	    REGION 180

	        REGION Displacement
	            #sFB_Displacement180(#sUDT_Interface_180);
	        END_REGION

	        REGION Conveyor

	            #sUDT_Handshake_180.RTR := TRUE;

	            #sFB_Conveyor_080(iUDT_ConveyorConfiguration := #iqUDT_Configuration."180".Conveyor,
	                              idi_PECEoSDistance := 0,
	                              idi_PECBoSDistance := 0,
	                              ii_ExternalSpeed := 0,
	                              ix_SafetyOk := #ix_SafetyOk,
	                              ix_24vOk := #ix_24vOk,
	                              ix_400vOk := #ix_400vOk,
	                              ix_HardwareOk := TRUE,
	                              ix_PECEoS := TRUE,
	                              ix_PECBoS := TRUE,
	                              ix_ReverseDirection := FALSE,
	                              ix_ExternalRequestDieBack := FALSE,
	                              ix_ExternalRequestHold := #sx_Hold180,
	                              ix_ResetEnergySave := FALSE,
	                              qUDT_HMIStatus => #iqUDT_WorkstationStatus."180".Conveyor,
	                              qUDT_Status => #iqUDT_WorkstationCommonStatus."180",
	                              iqUDT_EquipmentControl := #iqUDT_EquipmentControl,
	                              iqUDT_ConveyorCommand := #iqUDT_WorkstationCommands."180".Conveyor,
	                              iqUDT_ConveyorInterface := #sUDT_Interface_180,
	                              iqUDT_HandShakeUp := #sUDT_HandshakeUp_180,
	                              iqUDT_HandShake := #sUDT_Handshake_180,
	                              iqUDT_Statistics := #iqUDT_WorkstationStatistics."180".Conveyor);

	        END_REGION

	        REGION MCO

	            #sFB_MCOConveyLinxAixController_180(iUDT_AixConfig := #iqUDT_Configuration."180".MCO_M01,
	                                                iUDT_AixInputsModule := #iUDT_MotorInput170,
	                                                ix_24vOk := #ix_24vOk,
	                                                ix_SimulationModeActive := "DB_Memory".Simulation,
	                                                ii_MotorPositionId := 2,
	                                                qUDT_HMIStatus => #iqUDT_WorkstationStatus."180".MCO_M01,
	                                                iqUDT_AixOutputsModule := #iqUDT_MotorOutput170,
	                                                iqUDT_ConveyorInterface := #sUDT_Interface_180,
	                                                iqUDT_MCOStatistics := #iqUDT_WorkstationStatistics."180".MCO_M01);
	        END_REGION

	    END_REGION
	END_IF;
	REGION 210

	    REGION Displacement
	        #sFB_Displacement210(#sUDT_Interface_210);
	    END_REGION

	    REGION Tracking

	        #sFB_Tracking_210(iUDT_ConveyorCommonConfiguration := #iqUDT_Configuration."210".Conveyor.Common,
	                          iqa_TrackingData := #sa_TrackingArray_210,
	                          iqUDT_ConveyorInterface := #sUDT_Interface_210,
	                          iqUDT_HandshakeUp := #sUDT_HandshakeUp_210,
	                          iqUDT_Handshake := #sUDT_Handshake_210);

	    END_REGION

	    REGION EoS

	        #sFB_PECUpdate_210(iUDT_PECUpdateConfiguration := #iqUDT_Configuration."210".PEC_EoS,
	                           iUDT_ConveyorCommonConfiguration := #iqUDT_Configuration."210".Conveyor.Common,
	                           ix_PEC := NOT #iUDT_MotorInput210.AllSensorPortInputs.LeftSensor,
	                           ix_TeachingMode := FALSE,
	                           qUDT_Status => #iqUDT_WorkstationStatus."210".PEC_EoS,
	                           iqUDT_ConveyorInterface := #sUDT_Interface_210,
	                           iqUDT_UnknownGINRange := #iqUDT_UnknownGINRange,
	                           iqUDT_FifoHeader := "DB_FIFOLostGIN".Header,
	                           iqUDT_Statistics := #iqUDT_WorkstationStatistics."210".PEC_EoS,
	                           iqa_TrackingData := #sa_TrackingArray_210,
	                           iqa_FifoData := "DB_FIFOLostGIN".Data);

	    END_REGION

	    REGION Conveyor

	        #sFB_Conveyor_210(iUDT_ConveyorConfiguration := #iqUDT_Configuration."210".Conveyor,
	                          idi_PECEoSDistance := #iqUDT_Configuration."210".PEC_EoS.Distance,
	                          idi_PECBoSDistance := 0,
	                          ii_ExternalSpeed := 0,
	                          ix_SafetyOk := #ix_SafetyOk,
	                          ix_24vOk := #ix_24vOk,
	                          ix_400vOk := #ix_400vOk,
	                          ix_HardwareOk := TRUE,
	                          ix_PECEoS := #iqUDT_WorkstationStatus."210".PEC_EoS.PEC,
	                          ix_PECBoS := TRUE,
	                          ix_ReverseDirection := FALSE,
	                          ix_ExternalRequestDieBack := FALSE,
	                          ix_ExternalRequestHold := #sx_ReleaseBinHoldLeft OR #sx_ReleaseBinHoldRight OR NOT #sUDT_Handshake_210.RTR,
	                          ix_ResetEnergySave := FALSE,
	                          qUDT_HMIStatus => #iqUDT_WorkstationStatus."210".Conveyor,
	                          qUDT_Status => #iqUDT_WorkstationCommonStatus."210",
	                          iqUDT_EquipmentControl := #iqUDT_EquipmentControl,
	                          iqUDT_ConveyorCommand := #iqUDT_WorkstationCommands."210".Conveyor,
	                          iqUDT_ConveyorInterface := #sUDT_Interface_210,
	                          iqUDT_HandShakeUp := #sUDT_HandshakeUp_210,
	                          iqUDT_HandShake := #sUDT_Handshake_210,
	                          iqUDT_Statistics := #iqUDT_WorkstationStatistics."210".Conveyor);

	    END_REGION

	    REGION MCO

	        #sFB_MCOConveyLinxAixController_210(iUDT_AixConfig := #iqUDT_Configuration."210".MCO_M01,
	                                            iUDT_AixInputsModule := #iUDT_MotorInput210,
	                                            ix_24vOk := #ix_24vOk,
	                                            ix_SimulationModeActive := "DB_Memory".Simulation,
	                                            ii_MotorPositionId := 1,
	                                            qUDT_HMIStatus => #iqUDT_WorkstationStatus."210".MCO_M01,
	                                            iqUDT_AixOutputsModule := #iqUDT_MotorOutput210,
	                                            iqUDT_ConveyorInterface := #sUDT_Interface_210,
	                                            iqUDT_MCOStatistics := #iqUDT_WorkstationStatistics."210".MCO_M01);
	    END_REGION

	END_REGION

	REGION 220

	    REGION Displacement
	        #sFB_Displacement220(#sUDT_Interface_220);
	    END_REGION

	    REGION Tracking

	        #sFB_Tracking_220(iUDT_ConveyorCommonConfiguration := #iqUDT_Configuration."220".Conveyor.Common,
	                          iqa_TrackingData := #sa_TrackingArray_220,
	                          iqUDT_ConveyorInterface := #sUDT_Interface_220,
	                          iqUDT_HandshakeUp := #sUDT_Handshake_210,
	                          iqUDT_Handshake := #sUDT_Handshake_220);

	    END_REGION

	    REGION EoS

	        #sFB_PECUpdate_220(iUDT_PECUpdateConfiguration := #iqUDT_Configuration."220".PEC_EoS,
	                           iUDT_ConveyorCommonConfiguration := #iqUDT_Configuration."220".Conveyor.Common,
	                           ix_PEC := NOT #iUDT_MotorInput210.AllSensorPortInputs.RightSensor,
	                           ix_TeachingMode := FALSE,
	                           qUDT_Status => #iqUDT_WorkstationStatus."220".PEC_EoS,
	                           iqUDT_ConveyorInterface := #sUDT_Interface_220,
	                           iqUDT_UnknownGINRange := #iqUDT_UnknownGINRange,
	                           iqUDT_FifoHeader := "DB_FIFOLostGIN".Header,
	                           iqUDT_Statistics := #iqUDT_WorkstationStatistics."220".PEC_EoS,
	                           iqa_TrackingData := #sa_TrackingArray_220,
	                           iqa_FifoData := "DB_FIFOLostGIN".Data);




	    END_REGION

	    REGION Conveyor

	        #sFB_Conveyor_220(iUDT_ConveyorConfiguration := #iqUDT_Configuration."220".Conveyor,
	                          idi_PECEoSDistance := #iqUDT_Configuration."220".PEC_EoS.Distance,
	                          idi_PECBoSDistance := 0,
	                          ii_ExternalSpeed := 0,
	                          ix_SafetyOk := #ix_SafetyOk,
	                          ix_24vOk := #ix_24vOk,
	                          ix_400vOk := #ix_400vOk,
	                          ix_HardwareOk := TRUE,
	                          ix_PECEoS := #iqUDT_WorkstationStatus."220".PEC_EoS.PEC,
	                          ix_PECBoS := TRUE,
	                          ix_ReverseDirection := FALSE,
	                          ix_ExternalRequestDieBack := FALSE,
	                          ix_ExternalRequestHold := #sx_Hold220 OR #sx_ReleaseBinHoldLeft OR #sx_ReleaseBinHoldRight,
	                          ix_ResetEnergySave := FALSE,
	                          qUDT_HMIStatus => #iqUDT_WorkstationStatus."220".Conveyor,
	                          qUDT_Status => #iqUDT_WorkstationCommonStatus."220",
	                          iqUDT_EquipmentControl := #iqUDT_EquipmentControl,
	                          iqUDT_ConveyorCommand := #iqUDT_WorkstationCommands."220".Conveyor,
	                          iqUDT_ConveyorInterface := #sUDT_Interface_220,
	                          iqUDT_HandShakeUp := #sUDT_Handshake_210,
	                          iqUDT_HandShake := #sUDT_Handshake_220,
	                          iqUDT_Statistics := #iqUDT_WorkstationStatistics."220".Conveyor);

	    END_REGION

	    REGION MCO

	        #sFB_MCOConveyLinxAixController_220(iUDT_AixConfig := #iqUDT_Configuration."220".MCO_M01,
	                                            iUDT_AixInputsModule := #iUDT_MotorInput210,
	                                            ix_24vOk := #ix_24vOk,
	                                            ix_SimulationModeActive := "DB_Memory".Simulation,
	                                            ii_MotorPositionId := 2,
	                                            qUDT_HMIStatus => #iqUDT_WorkstationStatus."220".MCO_M01,
	                                            iqUDT_AixOutputsModule := #iqUDT_MotorOutput210,
	                                            iqUDT_ConveyorInterface := #sUDT_Interface_220,
	                                            iqUDT_MCOStatistics := #iqUDT_WorkstationStatistics."220".MCO_M01);
	    END_REGION


	END_REGION

	REGION 230

	    REGION Displacement
	        #sFB_Displacement230(#sUDT_Interface_230);
	    END_REGION

	    REGION Tracking

	        #sFB_Tracking_230(iUDT_ConveyorCommonConfiguration := #iqUDT_Configuration."230".Conveyor.Common,
	                          iqa_TrackingData := #sa_TrackingArray_230,
	                          iqUDT_ConveyorInterface := #sUDT_Interface_230,
	                          iqUDT_HandshakeUp := #sUDT_Handshake_220,
	                          iqUDT_Handshake := #sUDT_Handshake_230);

	    END_REGION

	    REGION EoS

	        #sFB_PECUpdate_230(iUDT_PECUpdateConfiguration := #iqUDT_Configuration."230".PEC_EoS,
	                           iUDT_ConveyorCommonConfiguration := #iqUDT_Configuration."230".Conveyor.Common,
	                           ix_PEC := NOT #iUDT_MotorInput230.AllSensorPortInputs.LeftSensor,
	                           ix_TeachingMode := FALSE,
	                           qUDT_Status => #iqUDT_WorkstationStatus."230".PEC_EoS,
	                           iqUDT_ConveyorInterface := #sUDT_Interface_230,
	                           iqUDT_UnknownGINRange := #iqUDT_UnknownGINRange,
	                           iqUDT_FifoHeader := "DB_FIFOLostGIN".Header,
	                           iqUDT_Statistics := #iqUDT_WorkstationStatistics."230".PEC_EoS,
	                           iqa_TrackingData := #sa_TrackingArray_230,
	                           iqa_FifoData := "DB_FIFOLostGIN".Data);




	    END_REGION

	    REGION Conveyor
	        #sUDT_Handshake_230.RTR := #sUDT_Handshake_230.RTR OR #iqUDT_WorkstationStatus."230".PEC_EoS.PEC;
	        #sFB_Conveyor_230(iUDT_ConveyorConfiguration := #iqUDT_Configuration."230".Conveyor,
	                          idi_PECEoSDistance := #iqUDT_Configuration."230".PEC_EoS.Distance,
	                          idi_PECBoSDistance := 0,
	                          ii_ExternalSpeed := 0,
	                          ix_SafetyOk := #ix_SafetyOk,
	                          ix_24vOk := #ix_24vOk,
	                          ix_400vOk := #ix_400vOk,
	                          ix_HardwareOk := TRUE,
	                          ix_PECEoS := #iqUDT_WorkstationStatus."230".PEC_EoS.PEC,
	                          ix_PECBoS := TRUE,
	                          ix_ReverseDirection := FALSE,
	                          ix_ExternalRequestDieBack := FALSE,
	                          ix_ExternalRequestHold := #sx_Hold230 OR #sx_ReleaseBinHoldLeft OR #sx_ReleaseBinHoldRight,
	                          ix_ResetEnergySave := FALSE,
	                          qUDT_HMIStatus => #iqUDT_WorkstationStatus."230".Conveyor,
	                          qUDT_Status => #iqUDT_WorkstationCommonStatus."230",
	                          iqUDT_EquipmentControl := #iqUDT_EquipmentControl,
	                          iqUDT_ConveyorCommand := #iqUDT_WorkstationCommands."230".Conveyor,
	                          iqUDT_ConveyorInterface := #sUDT_Interface_230,
	                          iqUDT_HandShakeUp := #sUDT_Handshake_220,
	                          iqUDT_HandShake := #sUDT_Handshake_230,
	                          iqUDT_Statistics := #iqUDT_WorkstationStatistics."230".Conveyor);

	    END_REGION

	    REGION MCO

	        #sFB_MCOConveyLinxAixController_230(iUDT_AixConfig := #iqUDT_Configuration."230".MCO_M01,
	                                            iUDT_AixInputsModule := #iUDT_MotorInput230,
	                                            ix_24vOk := #ix_24vOk,
	                                            ix_SimulationModeActive := "DB_Memory".Simulation,
	                                            ii_MotorPositionId := 1,
	                                            qUDT_HMIStatus => #iqUDT_WorkstationStatus."230".MCO_M01,
	                                            iqUDT_AixOutputsModule := #iqUDT_MotorOutput230,
	                                            iqUDT_ConveyorInterface := #sUDT_Interface_230,
	                                            iqUDT_MCOStatistics := #iqUDT_WorkstationStatistics."230".MCO_M01);
	    END_REGION

	END_REGION

	REGION 240

	    REGION Displacement
	        #sFB_Displacement240(#sUDT_Interface_240);
	    END_REGION

	    REGION MCO

	        #sFB_MCOConveyLinxAixController_240(iUDT_AixConfig := #iqUDT_Configuration."240".MCO_M01,
	                                            iUDT_AixInputsModule := #iUDT_MotorInput240,
	                                            ii_PositionSetpoint := #iqUDT_RATPositioning240.Lower.EndPosition,
	                                            ix_24vOk := #ix_24vOk,
	                                            ix_SimulationModeActive := "DB_Memory".Simulation,
	                                            ii_MotorPositionId := 1,
	                                            ix_StartPositioning := #iqUDT_RATPositioning240.Lower.Start,
	                                            ix_ResetPosition := #iqUDT_RATPositioning240.Lower.ResetPosition,
	                                            qUDT_HMIStatus => #iqUDT_WorkstationStatus."240".MCO_M01,
	                                            qx_Positioned => #iqUDT_RATPositioning240.Lower.Done,
	                                            iqUDT_AixOutputsModule := #iqUDT_MotorOutput240,
	                                            iqUDT_ConveyorInterface := #sUDT_Interface_240,
	                                            iqUDT_MCOStatistics := #iqUDT_WorkstationStatistics."240".MCO_M01);
	    END_REGION

	END_REGION

	REGION 241

	    REGION Displacement
	        #sFB_Displacement241(#sUDT_Interface_241);
	    END_REGION

	    REGION RAT

	        #sFB_RightAngledTransfer_241(iUDT_Configuration := #iqUDT_Configuration."241".RightAngledTransfer,
	                                     iUDT_LowerConveyorConfiguration := #iqUDT_Configuration."240".Conveyor,
	                                     iUDT_UpperConveyorConfiguration := #iqUDT_Configuration."241".Conveyor,
	                                     iUDT_PECConfiguration := #iqUDT_Configuration."240".PEC_EoS,
	                                     ii_DestinationA := #si_240DestinationA,
	                                     ii_DestinationB := #si_240DestinationB,
	                                     ii_DestinationC := #si_240DestinationC,
	                                     ii_DestinationD := #si_240DestinationD,
	                                     ix_HardwareOk := TRUE,
	                                     ix_400vOk := #ix_400vOk,
	                                     ix_24vOk := #ix_24vOk,
	                                     ix_SafetyOk := #ix_SafetyOk,
	                                     ix_AirPressureOk := #ix_AirPressureOk,
	                                     ix_SectionIsDown := #ix_SectionisDown241,
	                                     ix_SectionIsUp := #ix_SectionisUp241,
	                                     ix_ConveyorAAuto := #iqUDT_WorkstationCommonStatus."230".AutoON,
	                                     ix_ConveyorBAuto := #iqUDT_WorkstationCommonStatus."250".AutoON,
	                                     ix_ConveyorCAuto := #iqUDT_WorkstationCommonStatus."141".AutoON,
	                                     ix_ConveyorDAuto := #iqUDT_WorkstationCommonStatus."041".AutoON,
	                                     ix_PEC := #iUDT_MotorInput240.AllSensorPortInputs.LeftSensor,
	                                     ix_ExternalReceiveRequestA := NOT #iqUDT_WorkstationStatus."230".PEC_EoS.PEC AND #sx_Enable2X0In,
	                                     ix_ExternalReceiveRequestB := false,
	                                     ix_ExternalReceiveRequestC := #sFB_RightAngledTransfer_141.qx_ExternalSendRequestC,
	                                     ix_ExternalReceiveRequestD := #sFB_RightAngledTransfer_041.qx_ExternalSendRequestD,
	                                     ix_PECInfeedA := #iqUDT_WorkstationStatus."230".PEC_EoS.PEC,
	                                     ix_PECInfeedC := #iqUDT_WorkstationStatus."140".PEC_EoS.PEC,
	                                     ix_PECInfeedD := #iqUDT_WorkstationStatus."040".PEC_EoS.PEC,
	                                     qUDT_HMIRATStatus => #iqUDT_WorkstationStatus."241".RightAngledTransfer,
	                                     qUDT_HMIConveyorStatus => #iqUDT_WorkstationStatus."240".Conveyor,
	                                     qUDT_HMIPECStatus => #iqUDT_WorkstationStatus."240".PEC_EoS,
	                                     qUDT_RATStatus => #iqUDT_WorkstationCommonStatus."241",
	                                     qUDT_ConveyorStatus => #iqUDT_WorkstationCommonStatus."240",
	                                     qx_PopupControl => #qx_PopupControl241,
	                                     iqUDT_EquipmentControl := #iqUDT_EquipmentControl,
	                                     iqUDT_RATCommand := #iqUDT_WorkstationCommands."241".RightAngledTransfer,
	                                     iqUDT_ConveyorCommand := #iqUDT_WorkstationCommands."240".Conveyor,
	                                     iqUDT_RATStatistics := #iqUDT_WorkstationStatistics."241".RightAngledTransfer,
	                                     iqUDT_ConveyorStatistics := #iqUDT_WorkstationStatistics."240".Conveyor,
	                                     iqUDT_PECStatistics := #iqUDT_WorkstationStatistics."240".PEC_EoS,
	                                     iqUDT_HandShakeConveyorA := #sUDT_Handshake_230,
	                                     iqUDT_HandShakeConveyorB := #sUDT_Handshake_240,
	                                     iqUDT_HandShakeConveyorC := #sUDT_Handshake_241,
	                                     iqUDT_HandShakeConveyorD := #sUDT_Handshake_041,
	                                     iqUDT_LowerConveyorInterface := #sUDT_Interface_240,
	                                     iqUDT_UpperConveyorInterface := #sUDT_Interface_241,
	                                     iqUDT_RATPositioning := #iqUDT_RATPositioning240,
	                                     iqUDT_BladeStopEoSInterface := #tUDT_DummyBladeStop,
	                                     iqUDT_BladeStopBoSInterface := #tUDT_DummyBladeStop);

	    END_REGION

	    REGION MCO

	        #sFB_MCOConveyLinxAixController_241(iUDT_AixConfig := #iqUDT_Configuration."241".MCO_M01,
	                                            iUDT_AixInputsModule := #iUDT_MotorInput240,
	                                            ii_PositionSetpoint := #iqUDT_RATPositioning240.Upper.EndPosition,
	                                            ix_24vOk := #ix_24vOk,
	                                            ix_SimulationModeActive := "DB_Memory".Simulation,
	                                            ii_MotorPositionId := 2,
	                                            ix_StartPositioning := #iqUDT_RATPositioning240.Upper.Start,
	                                            ix_ResetPosition := #iqUDT_RATPositioning240.Upper.ResetPosition,
	                                            qUDT_HMIStatus => #iqUDT_WorkstationStatus."241".MCO_M01,
	                                            qx_Positioned => #iqUDT_RATPositioning240.Upper.Done,
	                                            iqUDT_AixOutputsModule := #iqUDT_MotorOutput240,
	                                            iqUDT_ConveyorInterface := #sUDT_Interface_241,
	                                            iqUDT_MCOStatistics := #iqUDT_WorkstationStatistics."241".MCO_M01);
	    END_REGION

	END_REGION

	REGION 250

	    REGION Displacement
	        #sFB_Displacement250(#sUDT_Interface_250);
	    END_REGION

	    REGION Tracking

	        #sFB_Tracking_250(iUDT_ConveyorCommonConfiguration := #iqUDT_Configuration."250".Conveyor.Common,
	                          iqa_TrackingData := #sa_TrackingArray_250,
	                          iqUDT_ConveyorInterface := #sUDT_Interface_250,
	                          iqUDT_HandshakeUp := #sUDT_Handshake_240,
	                          iqUDT_Handshake := #sUDT_Handshake_250);

	    END_REGION

	    REGION EoS

	        #sFB_PECUpdate_250(iUDT_PECUpdateConfiguration := #iqUDT_Configuration."250".PEC_EoS,
	                           iUDT_ConveyorCommonConfiguration := #iqUDT_Configuration."250".Conveyor.Common,
	                           ix_PEC := #iUDT_MotorInput250.AllSensorPortInputs.LeftSensor,
	                           ix_TeachingMode := FALSE,
	                           qUDT_Status => #iqUDT_WorkstationStatus."250".PEC_EoS,
	                           iqUDT_ConveyorInterface := #sUDT_Interface_250,
	                           iqUDT_UnknownGINRange := #iqUDT_UnknownGINRange,
	                           iqUDT_FifoHeader := "DB_FIFOLostGIN".Header,
	                           iqUDT_Statistics := #iqUDT_WorkstationStatistics."250".PEC_EoS,
	                           iqa_TrackingData := #sa_TrackingArray_250,
	                           iqa_FifoData := "DB_FIFOLostGIN".Data);




	    END_REGION

	    REGION Conveyor

	        #sFB_Conveyor_250(iUDT_ConveyorConfiguration := #iqUDT_Configuration."250".Conveyor,
	                          idi_PECEoSDistance := 0,
	                          idi_PECBoSDistance := 0,
	                          ii_ExternalSpeed := 0,
	                          ix_SafetyOk := #ix_SafetyOk,
	                          ix_24vOk := #ix_24vOk,
	                          ix_400vOk := #ix_400vOk,
	                          ix_HardwareOk := TRUE,
	                          ix_PECEoS := #iqUDT_WorkstationStatus."250".PEC_EoS.PEC,
	                          ix_PECBoS := TRUE,
	                          ix_ReverseDirection := FALSE,
	                          ix_ExternalRequestDieBack := FALSE,
	                          ix_ExternalRequestHold := FALSE,
	                          ix_ResetEnergySave := FALSE,
	                          qUDT_HMIStatus => #iqUDT_WorkstationStatus."250".Conveyor,
	                          qUDT_Status => #iqUDT_WorkstationCommonStatus."250",
	                          iqUDT_EquipmentControl := #iqUDT_EquipmentControl,
	                          iqUDT_ConveyorCommand := #iqUDT_WorkstationCommands."250".Conveyor,
	                          iqUDT_ConveyorInterface := #sUDT_Interface_250,
	                          iqUDT_HandShakeUp := #sUDT_Handshake_240,
	                          iqUDT_HandShake := #sUDT_Handshake_250,
	                          iqUDT_Statistics := #iqUDT_WorkstationStatistics."250".Conveyor);

	    END_REGION

	    REGION MCO

	        #sFB_MCOConveyLinxAixController_250(iUDT_AixConfig := #iqUDT_Configuration."250".MCO_M01,
	                                            iUDT_AixInputsModule := #iUDT_MotorInput250,
	                                            ix_24vOk := #ix_24vOk,
	                                            ix_SimulationModeActive := "DB_Memory".Simulation,
	                                            ii_MotorPositionId := 1,
	                                            qUDT_HMIStatus => #iqUDT_WorkstationStatus."250".MCO_M01,
	                                            iqUDT_AixOutputsModule := #iqUDT_MotorOutput250,
	                                            iqUDT_ConveyorInterface := #sUDT_Interface_250,
	                                            iqUDT_MCOStatistics := #iqUDT_WorkstationStatistics."250".MCO_M01);
	    END_REGION

	END_REGION

	REGION 260

	    REGION Displacement
	        #sFB_Displacement260(#sUDT_Interface_260);
	    END_REGION

	    REGION Tracking

	        #sFB_Tracking_260(iUDT_ConveyorCommonConfiguration := #iqUDT_Configuration."260".Conveyor.Common,
	                          iqa_TrackingData := #sa_TrackingArray_260,
	                          iqUDT_ConveyorInterface := #sUDT_Interface_260,
	                          iqUDT_HandshakeUp := #sUDT_Handshake_250,
	                          iqUDT_Handshake := #sUDT_Handshake_260);

	    END_REGION

	    REGION EoS

	        #sFB_PECUpdate_260(iUDT_PECUpdateConfiguration := #iqUDT_Configuration."260".PEC_EoS,
	                           iUDT_ConveyorCommonConfiguration := #iqUDT_Configuration."260".Conveyor.Common,
	                           ix_PEC := #iUDT_MotorInput250.AllSensorPortInputs.RightSensor,
	                           ix_TeachingMode := FALSE,
	                           qUDT_Status => #iqUDT_WorkstationStatus."260".PEC_EoS,
	                           iqUDT_ConveyorInterface := #sUDT_Interface_260,
	                           iqUDT_UnknownGINRange := #iqUDT_UnknownGINRange,
	                           iqUDT_FifoHeader := "DB_FIFOLostGIN".Header,
	                           iqUDT_Statistics := #iqUDT_WorkstationStatistics."260".PEC_EoS,
	                           iqa_TrackingData := #sa_TrackingArray_260,
	                           iqa_FifoData := "DB_FIFOLostGIN".Data);




	    END_REGION

	    REGION Conveyor

	        #sFB_Conveyor_260(iUDT_ConveyorConfiguration := #iqUDT_Configuration."260".Conveyor,
	                          idi_PECEoSDistance := 0,
	                          idi_PECBoSDistance := 0,
	                          ii_ExternalSpeed := 0,
	                          ix_SafetyOk := #ix_SafetyOk,
	                          ix_24vOk := #ix_24vOk,
	                          ix_400vOk := #ix_400vOk,
	                          ix_HardwareOk := TRUE,
	                          ix_PECEoS := #iqUDT_WorkstationStatus."260".PEC_EoS.PEC,
	                          ix_PECBoS := TRUE,
	                          ix_ReverseDirection := FALSE,
	                          ix_ExternalRequestDieBack := FALSE,
	                          ix_ExternalRequestHold := FALSE,
	                          ix_ResetEnergySave := FALSE,
	                          qUDT_HMIStatus => #iqUDT_WorkstationStatus."260".Conveyor,
	                          qUDT_Status => #iqUDT_WorkstationCommonStatus."260",
	                          iqUDT_EquipmentControl := #iqUDT_EquipmentControl,
	                          iqUDT_ConveyorCommand := #iqUDT_WorkstationCommands."260".Conveyor,
	                          iqUDT_ConveyorInterface := #sUDT_Interface_260,
	                          iqUDT_HandShakeUp := #sUDT_Handshake_250,
	                          iqUDT_HandShake := #sUDT_Handshake_260,
	                          iqUDT_Statistics := #iqUDT_WorkstationStatistics."260".Conveyor);

	    END_REGION

	    REGION MCO

	        #sFB_MCOConveyLinxAixController_260(iUDT_AixConfig := #iqUDT_Configuration."260".MCO_M01,
	                                            iUDT_AixInputsModule := #iUDT_MotorInput250,
	                                            ix_24vOk := #ix_24vOk,
	                                            ix_SimulationModeActive := "DB_Memory".Simulation,
	                                            ii_MotorPositionId := 2,
	                                            qUDT_HMIStatus => #iqUDT_WorkstationStatus."260".MCO_M01,
	                                            iqUDT_AixOutputsModule := #iqUDT_MotorOutput250,
	                                            iqUDT_ConveyorInterface := #sUDT_Interface_260,
	                                            iqUDT_MCOStatistics := #iqUDT_WorkstationStatistics."260".MCO_M01);
	    END_REGION

	END_REGION

	REGION 270

	    REGION Displacement
	        #sFB_Displacement270(#sUDT_Interface_270);
	    END_REGION

	    REGION Tracking

	        #sFB_Tracking_270(iUDT_ConveyorCommonConfiguration := #iqUDT_Configuration."270".Conveyor.Common,
	                          iqa_TrackingData := #sa_TrackingArray_270,
	                          iqUDT_ConveyorInterface := #sUDT_Interface_270,
	                          iqUDT_HandshakeUp := #sUDT_Handshake_260,
	                          iqUDT_Handshake := #iqUDT_HandshakeDownstream270);

	    END_REGION

	    REGION EoS

	        #sFB_PECUpdate_270(iUDT_PECUpdateConfiguration := #iqUDT_Configuration."270".PEC_EoS,
	                           iUDT_ConveyorCommonConfiguration := #iqUDT_Configuration."270".Conveyor.Common,
	                           ix_PEC := #iUDT_MotorInput270.AllSensorPortInputs.LeftSensor,
	                           ix_TeachingMode := FALSE,
	                           qUDT_Status => #iqUDT_WorkstationStatus."270".PEC_EoS,
	                           iqUDT_ConveyorInterface := #sUDT_Interface_270,
	                           iqUDT_UnknownGINRange := #iqUDT_UnknownGINRange,
	                           iqUDT_FifoHeader := "DB_FIFOLostGIN".Header,
	                           iqUDT_Statistics := #iqUDT_WorkstationStatistics."270".PEC_EoS,
	                           iqa_TrackingData := #sa_TrackingArray_270,
	                           iqa_FifoData := "DB_FIFOLostGIN".Data);

	    END_REGION

	    REGION Conveyor

	        #iqUDT_HandshakeDownstream270.RTR := #iqUDT_HandshakeDownstream270.RTR OR #iqUDT_WorkstationStatus."270".PEC_EoS.PEC;

	        #sFB_Conveyor_270(iUDT_ConveyorConfiguration := #iqUDT_Configuration."270".Conveyor,
	                          idi_PECEoSDistance := #iqUDT_Configuration."270".PEC_EoS.Distance,
	                          idi_PECBoSDistance := 0,
	                          ii_ExternalSpeed := 0,
	                          ix_SafetyOk := #ix_SafetyOk,
	                          ix_24vOk := #ix_24vOk,
	                          ix_400vOk := #ix_400vOk,
	                          ix_HardwareOk := TRUE,
	                          ix_PECEoS := #iqUDT_WorkstationStatus."270".PEC_EoS.PEC,
	                          ix_PECBoS := TRUE,
	                          ix_ReverseDirection := FALSE,
	                          ix_ExternalRequestDieBack := FALSE,
	                          ix_ExternalRequestHold := FALSE,
	                          ix_ResetEnergySave := FALSE,
	                          qUDT_HMIStatus => #iqUDT_WorkstationStatus."270".Conveyor,
	                          qUDT_Status => #iqUDT_WorkstationCommonStatus."270",
	                          iqUDT_EquipmentControl := #iqUDT_EquipmentControl,
	                          iqUDT_ConveyorCommand := #iqUDT_WorkstationCommands."270".Conveyor,
	                          iqUDT_ConveyorInterface := #sUDT_Interface_270,
	                          iqUDT_HandShakeUp := #sUDT_Handshake_260,
	                          iqUDT_HandShake := #iqUDT_HandshakeDownstream270,
	                          iqUDT_Statistics := #iqUDT_WorkstationStatistics."270".Conveyor);

	    END_REGION

	    REGION MCO

	        #sFB_MCOConveyLinxAixController_270(iUDT_AixConfig := #iqUDT_Configuration."270".MCO_M01,
	                                            iUDT_AixInputsModule := #iUDT_MotorInput270,
	                                            ix_24vOk := #ix_24vOk,
	                                            ix_SimulationModeActive := "DB_Memory".Simulation,
	                                            ii_MotorPositionId := 1,
	                                            qUDT_HMIStatus => #iqUDT_WorkstationStatus."270".MCO_M01,
	                                            iqUDT_AixOutputsModule := #iqUDT_MotorOutput270,
	                                            iqUDT_ConveyorInterface := #sUDT_Interface_270,
	                                            iqUDT_MCOStatistics := #iqUDT_WorkstationStatistics."270".MCO_M01);
	    END_REGION

	END_REGION

END_FUNCTION_BLOCK

FUNCTION_BLOCK "FB_PushUpDivert"
TITLE = FB_PushUpDivert
{ S7_Optimized_Access := 'TRUE' }
VERSION : 0.1
// ATTRIBUTES
// AUTO_NUMBER = True
// BLOCK_NUMBER = 199
// END_ATTRIBUTES
//Function to control a divert left/right/straight. A product is diverted based on GIN data. A conveyor, part of the diverter, will move up or down to change the direction. Moving up and down control is done by this block.
   VAR_INPUT
      iUDT_DivertConfiguration { ExternalAccessible := 'False'; ExternalVisible := 'False'; ExternalWritable := 'False'} : "UDT_PushUpDivertConfiguration";   // Configuration structure
      ii_Gin { ExternalAccessible := 'False'; ExternalVisible := 'False'; ExternalWritable := 'False'} : Int;   // Gin found by position block
      ii_DisplacementLower { ExternalAccessible := 'False'; ExternalVisible := 'False'; ExternalWritable := 'False'} : Int;   // Actual displacement of the lower conveyor
      ii_DisplacementUpper { ExternalAccessible := 'False'; ExternalVisible := 'False'; ExternalWritable := 'False'} : Int;   // Actual displacement of the upper conveyor
      ix_AirPressureOk { ExternalAccessible := 'False'; ExternalVisible := 'False'; ExternalWritable := 'False'} : Bool;   // Air pressure circuit healthy
      ix_SafetyOk { ExternalAccessible := 'False'; ExternalVisible := 'False'; ExternalWritable := 'False'} : Bool;   // TRUE when safety is ok
      ix_24vOk { ExternalAccessible := 'False'; ExternalVisible := 'False'; ExternalWritable := 'False'} : Bool;   // TRUE when 24VDC is healthy
      ix_400vOk { ExternalAccessible := 'False'; ExternalVisible := 'False'; ExternalWritable := 'False'} : Bool;   // TRUE when 400VAC is healthy
      ix_HardwareOk { ExternalAccessible := 'False'; ExternalVisible := 'False'; ExternalWritable := 'False'} : Bool;   // TRUE when  hardware is Ok
      ix_PecTrigger { ExternalAccessible := 'False'; ExternalVisible := 'False'; ExternalWritable := 'False'} : Bool;   // TRUE when trigger is not occupied
      ix_PECLeft { ExternalAccessible := 'False'; ExternalVisible := 'False'; ExternalWritable := 'False'} : Bool;   // TRUE when left outfeed PEC is not occupied
      ix_PECRight { ExternalAccessible := 'False'; ExternalVisible := 'False'; ExternalWritable := 'False'} : Bool;   // TRUE when right outfeed PEC is not occupied
      ix_SectionIsUp { ExternalAccessible := 'False'; ExternalVisible := 'False'; ExternalWritable := 'False'} : Bool;   // TRUE when section is up
      ix_SectionIsDown { ExternalAccessible := 'False'; ExternalVisible := 'False'; ExternalWritable := 'False'} : Bool;   // TRUE when section is down
   END_VAR

   VAR_OUTPUT
      qUDT_HMIStatus { ExternalAccessible := 'False'; ExternalVisible := 'False'; ExternalWritable := 'False'} : "UDT_PushUpDivertStatus";   // HMI status structure
      qUDT_Status { ExternalAccessible := 'False'; ExternalVisible := 'False'; ExternalWritable := 'False'} : "UDT_CommonStatus";   // Common status structure
      qUDT_LowerConveyorInterface { ExternalAccessible := 'False'; ExternalVisible := 'False'; ExternalWritable := 'False'} : Struct   // Interface lower conveyor
         Hold { ExternalAccessible := 'False'; ExternalVisible := 'False'; ExternalWritable := 'False'} : Bool;   // Hold the conveyor
         RunFwd { ExternalAccessible := 'False'; ExternalVisible := 'False'; ExternalWritable := 'False'} : Bool;   // Run conveyor forward
         RunRvs { ExternalAccessible := 'False'; ExternalVisible := 'False'; ExternalWritable := 'False'} : Bool;   // Run conveyor reverse
      END_STRUCT;
      qUDT_UpperConveyorInterface { ExternalAccessible := 'False'; ExternalVisible := 'False'; ExternalWritable := 'False'} : Struct   // Interface upper conveyor
         Hold { ExternalAccessible := 'False'; ExternalVisible := 'False'; ExternalWritable := 'False'} : Bool;   // Hold the conveyor
         RunFwd { ExternalAccessible := 'False'; ExternalVisible := 'False'; ExternalWritable := 'False'} : Bool;   // Run conveyor forward
         RunRvs { ExternalAccessible := 'False'; ExternalVisible := 'False'; ExternalWritable := 'False'} : Bool;   // Run conveyor reverse
      END_STRUCT;
      qx_SectionUp { ExternalAccessible := 'False'; ExternalVisible := 'False'; ExternalWritable := 'False'} : Bool;   // Output to control section up
      qx_SectionDown { ExternalAccessible := 'False'; ExternalVisible := 'False'; ExternalWritable := 'False'} : Bool;   // Output to control section down
   END_VAR

   VAR_IN_OUT
      iqa_TrackingMainData : Array[*] of Int;   // Data tracking main conveyor
      iqUDT_EquipmentControl : "UDT_EquipmentControl";   // Equipment control structure
      iqUDT_DivertCommand : "UDT_PushUpDivertCommand";   // Conveyor command stucture
      iqUDT_Statistics : "UDT_ConveyorStatistics";   // Statistics structure
      iqUDT_HandShakeLowerConveyor : "UDT_ConveyorHandshake";
      iqUDT_HandShakeUpperConveyor : "UDT_ConveyorHandshake";
      iqUDT_HandShakeLeftConveyor : "UDT_ConveyorHandshake";   // Handshake structure in forward direction left
      iqUDT_HandShakerightConveyor : "UDT_ConveyorHandshake";   // Handshake structure in reverse direction right
      iqi_RequestedPosition { ExternalAccessible := 'False'; ExternalVisible := 'False'; ExternalWritable := 'False'} : Int;   // Handshake requested position from destination block
   END_VAR

   VAR
      sUDT_Status { ExternalAccessible := 'False'; ExternalVisible := 'False'; ExternalWritable := 'False'; S7_SetPoint := 'False'} : "UDT_CommonStatus";   // Common status structure
      sFB_PECTriggerOnOffDelay { ExternalAccessible := 'False'; ExternalVisible := 'False'; ExternalWritable := 'False'; S7_SetPoint := 'False'} : "FB_TimerOnOffDelay";   // Timer to filter PEC signal
      sFB_PECLeftOnOffDelay { ExternalAccessible := 'False'; ExternalVisible := 'False'; ExternalWritable := 'False'; S7_SetPoint := 'False'} : "FB_TimerOnOffDelay";   // Timer to filter PEC signal
      sFB_PECRightOnOffDelay { ExternalAccessible := 'False'; ExternalVisible := 'False'; ExternalWritable := 'False'; S7_SetPoint := 'False'} : "FB_TimerOnOffDelay";   // Timer to filter PEC signal
      sFB_UpMonitor { ExternalAccessible := 'False'; ExternalVisible := 'False'; ExternalWritable := 'False'; S7_SetPoint := 'False'} : "FB_TimerOnOffDelay";   // Timer to monitor divert took too long to move to upper position
      sFB_DownMonitor { ExternalAccessible := 'False'; ExternalVisible := 'False'; ExternalWritable := 'False'; S7_SetPoint := 'False'} : "FB_TimerOnOffDelay";
      sR_TRIG_ManualMode {InstructionName := 'R_TRIG'; LibVersion := '1.0'; ExternalAccessible := 'False'; ExternalVisible := 'False'; ExternalWritable := 'False'; S7_SetPoint := 'False'} : R_TRIG;   // Rising edge trigger manual mode
      sF_TRIG_ManualMode {InstructionName := 'F_TRIG'; LibVersion := '1.0'; ExternalAccessible := 'False'; ExternalVisible := 'False'; ExternalWritable := 'False'; S7_SetPoint := 'False'} : F_TRIG;   // Falling edge trigger manual mode
      sR_TRIG_PrestartManual {InstructionName := 'R_TRIG'; LibVersion := '1.0'; ExternalAccessible := 'False'; ExternalVisible := 'False'; ExternalWritable := 'False'; S7_SetPoint := 'False'} : R_TRIG;   // Rising edge of manual prestart
      sR_TRIG_RunManual {InstructionName := 'R_TRIG'; LibVersion := '1.0'; ExternalAccessible := 'False'; ExternalVisible := 'False'; ExternalWritable := 'False'; S7_SetPoint := 'False'} : R_TRIG;   // Rising edge run conveyor in manual mode
      sR_TRIG_ManualGoUp {InstructionName := 'R_TRIG'; LibVersion := '1.0'; ExternalAccessible := 'False'; ExternalVisible := 'False'; ExternalWritable := 'False'; S7_SetPoint := 'False'} : R_TRIG;   // Rising edge run conveyor in manual mode
      sR_TRIG_ManualGoDown {InstructionName := 'R_TRIG'; LibVersion := '1.0'; ExternalAccessible := 'False'; ExternalVisible := 'False'; ExternalWritable := 'False'; S7_SetPoint := 'False'} : R_TRIG;   // Rising edge trigger manual jog
      sF_TRIG_Jog {InstructionName := 'F_TRIG'; LibVersion := '1.0'; ExternalAccessible := 'False'; ExternalVisible := 'False'; ExternalWritable := 'False'; S7_SetPoint := 'False'} : F_TRIG;   // Falling edge trigger manual mode jog
      sR_TRIG_PECLeft {InstructionName := 'R_TRIG'; LibVersion := '1.0'; ExternalAccessible := 'False'; ExternalVisible := 'False'; ExternalWritable := 'False'; S7_SetPoint := 'False'} : R_TRIG;   // Rising edge trigger PEC left outfeed side
      sR_TRIG_PECRight {InstructionName := 'R_TRIG'; LibVersion := '1.0'; ExternalAccessible := 'False'; ExternalVisible := 'False'; ExternalWritable := 'False'; S7_SetPoint := 'False'} : R_TRIG;   // Rising edge trigger PEC right outfeed side
      sR_TRIG_DeviceUpTime {InstructionName := 'R_TRIG'; LibVersion := '1.0'; ExternalAccessible := 'False'; ExternalVisible := 'False'; ExternalWritable := 'False'; S7_SetPoint := 'False'} : R_TRIG;   // Rising edge trigger device up time
      sR_TRIG_DeviceStopped {InstructionName := 'R_TRIG'; LibVersion := '1.0'; ExternalAccessible := 'False'; ExternalVisible := 'False'; ExternalWritable := 'False'; S7_SetPoint := 'False'} : R_TRIG;   // Rising edge of stop
      sR_TRIG_DeviceDownTime {InstructionName := 'R_TRIG'; LibVersion := '1.0'; ExternalAccessible := 'False'; ExternalVisible := 'False'; ExternalWritable := 'False'; S7_SetPoint := 'False'} : R_TRIG;   // Rising edge trigger device down
      sdi_Divertposition { ExternalAccessible := 'False'; ExternalVisible := 'False'; ExternalWritable := 'False'} : DInt;   // Calculated: position in tracking to initiate divert
      si_Gin { ExternalAccessible := 'False'; ExternalVisible := 'False'; ExternalWritable := 'False'} : Int;   // New GIN found
      si_length { ExternalAccessible := 'False'; ExternalVisible := 'False'; ExternalWritable := 'False'} : Int;   // Length of the parcel
      si_Direction { ExternalAccessible := 'False'; ExternalVisible := 'False'; ExternalWritable := 'False'} : Int;   // Direction from decisionpoint
      si_OldDirection { ExternalAccessible := 'False'; ExternalVisible := 'False'; ExternalWritable := 'False'} : Int;   // Last direction from decisionpoint
      si_Position { ExternalAccessible := 'False'; ExternalVisible := 'False'; ExternalWritable := 'False'} : Int;   // Position counter
      sx_PECTriggerFiltered { ExternalAccessible := 'False'; ExternalVisible := 'False'; ExternalWritable := 'False'} : Bool;   // Signal filtered with on and off delay
      sx_PECLeftFiltered { ExternalAccessible := 'False'; ExternalVisible := 'False'; ExternalWritable := 'False'} : Bool;   // Signal filtered with on and off delay
      sx_PECRightFiltered { ExternalAccessible := 'False'; ExternalVisible := 'False'; ExternalWritable := 'False'} : Bool;   // Signal filtered with on and off delay
      sx_Active { ExternalAccessible := 'False'; ExternalVisible := 'False'; ExternalWritable := 'False'} : Bool;   // Divert sequence is activated for parcel
      sx_MoveSectionUp { ExternalAccessible := 'False'; ExternalVisible := 'False'; ExternalWritable := 'False'} : Bool;   // Step move divert to upper position
      sx_MoveSectionDown { ExternalAccessible := 'False'; ExternalVisible := 'False'; ExternalWritable := 'False'} : Bool;   // Step move divert to lower position
      sx_TransportActive { ExternalAccessible := 'False'; ExternalVisible := 'False'; ExternalWritable := 'False'} : Bool;   // Step transport is activated
      sx_Ready { ExternalAccessible := 'False'; ExternalVisible := 'False'; ExternalWritable := 'False'} : Bool;   // Conveyor Ready to operate in Automatic mode
      sx_AutomaticActive { ExternalAccessible := 'False'; ExternalVisible := 'False'; ExternalWritable := 'False'} : Bool;   // Running in automatic
      sx_PreStartManual { ExternalAccessible := 'False'; ExternalVisible := 'False'; ExternalWritable := 'False'} : Bool;   // Pre conditions to run conveyor in manual mode
      sx_ManualModeActive { ExternalAccessible := 'False'; ExternalVisible := 'False'; ExternalWritable := 'False'} : Bool;   // Manual mode active
      sx_ManualRunning { ExternalAccessible := 'False'; ExternalVisible := 'False'; ExternalWritable := 'False'} : Bool;   // Conveyor running in manual mode
      sx_ManualGoUp { ExternalAccessible := 'False'; ExternalVisible := 'False'; ExternalWritable := 'False'} : Bool;   // Manual control go Up
      sx_ManualGoDown { ExternalAccessible := 'False'; ExternalVisible := 'False'; ExternalWritable := 'False'} : Bool;   // Manual control go down
      sx_ManUP { ExternalAccessible := 'False'; ExternalVisible := 'False'; ExternalWritable := 'False'} : Bool;   // Manual go up
      sx_ManDown { ExternalAccessible := 'False'; ExternalVisible := 'False'; ExternalWritable := 'False'} : Bool;   // Manual go down
      sx_ConfigurationError { ExternalAccessible := 'False'; ExternalVisible := 'False'; ExternalWritable := 'False'} : Bool;   // Commissioning: configuration of parameters is wrong
      sx_LeftRequest { ExternalAccessible := 'False'; ExternalVisible := 'False'; ExternalWritable := 'False'} : Bool;   // Request left outfeed position for actual parcel
      sx_RightRequest { ExternalAccessible := 'False'; ExternalVisible := 'False'; ExternalWritable := 'False'} : Bool;   // Request right outfeed position for actual parcel
      sx_DivertUpRunTimeErr { ExternalAccessible := 'False'; ExternalVisible := 'False'; ExternalWritable := 'False'} : Bool;   // It is taking too long to move divert up
      sx_DivertDownRunTimeErr { ExternalAccessible := 'False'; ExternalVisible := 'False'; ExternalWritable := 'False'} : Bool;   // It is taking too long to move divert down
      sx_UpTime { ExternalAccessible := 'False'; ExternalVisible := 'False'; ExternalWritable := 'False'} : Bool;   // Device is up
      sx_DownTime { ExternalAccessible := 'False'; ExternalVisible := 'False'; ExternalWritable := 'False'} : Bool;   // Device is down
      sx_StoppedTime { ExternalAccessible := 'False'; ExternalVisible := 'False'; ExternalWritable := 'False'} : Bool;   // Device is stopped
   END_VAR

   VAR_TEMP
      ta_ConfigErr : Array[0..10] of Bool;
   END_VAR


BEGIN
	(*
	----------------------------------------------------------------------------------------

	Version history:
	Date        | Version   | Author        | Remark
	----------------------------------------------------------------------------------------
	13/02/2023  | 1.0       | F.Baten       | Initial version
	*)

	REGION 1 - Initial
	    REGION 1.1 - First PLC cycle

	        IF "DB_Memory".FirstScan
	        THEN
	            #sx_AutomaticActive := FALSE;                               // switch of automatic active

	        END_IF;

	    END_REGION

	    REGION 1.2 - Triggers

	        // Rising edge trigger manual mode
	        #sR_TRIG_ManualMode(CLK := #iqUDT_DivertCommand.ManualMode
	                            OR #iqUDT_EquipmentControl.Command.ManualMode);

	        // Falling edge trigger manual mode
	        #sF_TRIG_ManualMode(CLK := #iqUDT_DivertCommand.ManualMode
	                            OR #iqUDT_EquipmentControl.Command.ManualMode);

	        // Rising edge trigger PEC Left side
	        #sR_TRIG_PECLeft(CLK := #sx_PECLeftFiltered);

	        // Rising edge trigger PEC right side
	        #sR_TRIG_PECRight(CLK := #sx_PECRightFiltered);

	        // Rising edge trigger to start in manual mode
	        #sR_TRIG_RunManual(CLK := #iqUDT_DivertCommand.ManualStartStop);

	        // Rising edge trigger to go up in manual mode
	        #sR_TRIG_ManualGoUp(CLK := #iqUDT_DivertCommand.ManualUp);

	        // Rising edge trigger to go down in manual mode
	        #sR_TRIG_ManualGoDown(CLK := #iqUDT_DivertCommand.ManualDown);

	        // Rising edge equipment uptime
	        #sR_TRIG_DeviceUpTime(CLK := #sx_UpTime);

	        //Rising edge equipment stopped
	        #sR_TRIG_DeviceStopped(CLK := #sx_StoppedTime);

	        // Rising edge equipment conveyor downtime
	        #sR_TRIG_DeviceDownTime(CLK := #sx_DownTime);
	    END_REGION

	    REGION 1.3 - Timers
	        // Statement section REGION
	        #sFB_PECTriggerOnOffDelay(iudi_OnDelayTime := #iUDT_DivertConfiguration.PECTriggerTimeOnDelay,      // Off delay time to filter PEC signal
	                                  iudi_OffDelayTime := #iUDT_DivertConfiguration.PECTriggerTimeOffDelay,    // On delay time to filter PEC signal
	                                  ix_SignalToDelay := #ix_PecTrigger,                                       // PEC input signal
	                                  ix_Enable := TRUE,
	                                  qx_DelayedSignal => #sx_PECTriggerFiltered);                              // PEC signal filtered

	        #sFB_PECLeftOnOffDelay(iudi_OnDelayTime := #iUDT_DivertConfiguration.PECLeftTimeOnDelay,            // Off delay time to filter PEC signal
	                               iudi_OffDelayTime := #iUDT_DivertConfiguration.PECLeftTimeOffDelay,          // On delay time to filter PEC signal
	                               ix_SignalToDelay := #ix_PECLeft,                                             // PEC input signal
	                               ix_Enable := TRUE,
	                               qx_DelayedSignal => #sx_PECLeftFiltered);                                    // PEC signal filtered

	        #sFB_PECRightOnOffDelay(iudi_OnDelayTime := #iUDT_DivertConfiguration.PECRightTimeOnDelay,          // Off delay time to filter PEC signal
	                                iudi_OffDelayTime := #iUDT_DivertConfiguration.PECRightTimeOffDelay,        // On delay time to filter PEC signal
	                                ix_SignalToDelay := #ix_PECRight,                                           // PEC input signal
	                                ix_Enable := TRUE,
	                                qx_DelayedSignal => #sx_PECRightFiltered);                                  // PEC signal filtered

	        #sFB_UpMonitor(iudi_OnDelayTime := #iUDT_DivertConfiguration.DivertMonitorUpOnDelay,                // Off delay time
	                       iudi_OffDelayTime := #iUDT_DivertConfiguration.DivertMonitorUPOffDelay,              // On delay time
	                       ix_SignalToDelay := #sx_AutomaticActive
	                       AND #sx_MoveSectionUp
	                       AND NOT #ix_SectionIsUp,                                                             // input signal
	                       ix_Enable := TRUE,
	                       qx_DelayedSignal => #sx_DivertUpRunTimeErr);                                         // signal filtered

	        #sFB_DownMonitor(iudi_OnDelayTime := #iUDT_DivertConfiguration.DivertMonitorDownOnDelay,            // Off delay time to filter PEC signal
	                         iudi_OffDelayTime := #iUDT_DivertConfiguration.DivertMonitorDownOffDelay,          // On delay time to filter PEC signal
	                         ix_SignalToDelay := #sx_AutomaticActive
	                         AND #sx_MoveSectionDown
	                         AND NOT #ix_SectionIsDown,                                                         // PEC input signal
	                         ix_Enable := TRUE,
	                         qx_DelayedSignal => #sx_DivertDownRunTimeErr);                                     // PEC signal filtered

	    END_REGION

	    REGION 1.4 - Conditions Up - Down - Stopped
	        //Used for statistics

	        #sx_UpTime := (#sx_AutomaticActive                              // Automatic active
	        AND #sx_Ready);                                                 // Ready active

	        #sx_DownTime := (NOT #sx_ManualModeActive                       // Not in manual mode
	        AND #sUDT_Status.Error                                          // in error
	        AND NOT #sx_Ready);                                             // Conveyor not ready

	        #sx_StoppedTime := (NOT #sx_AutomaticActive AND #sx_Ready);

	    END_REGION

	END_REGION

	REGION 2 - Errors

	    REGION 2.1 - Reset errors

	        IF #iqUDT_EquipmentControl.Command.Reset                        // Reset
	        THEN

	            IF #qUDT_HMIStatus.Specific.ErrRuntime                      // It took too long to move divert up or down
	            THEN

	                #qUDT_HMIStatus.Specific.ErrRuntime := FALSE;           // reset error

	            END_IF;

	            IF #qUDT_HMIStatus.Specific.ErrAirpressureNotOk             // Airpressure is not ok
	            THEN

	                #qUDT_HMIStatus.Specific.ErrAirpressureNotOk := FALSE;  // reset error

	            END_IF;

	            IF #qUDT_HMIStatus.Specific.ErrOverrun                      // It took too long to move divert up or down
	            THEN

	                #qUDT_HMIStatus.Specific.ErrOverrun := FALSE;           // reset error

	            END_IF;

	            IF #sx_DivertUpRunTimeErr                                   // It took too long to move up
	                AND #sx_MoveSectionUp                                   // It took too long to move down
	            THEN
	                #si_Gin := 0;                                           // Reset the GIN to write
	                #sx_MoveSectionDown := TRUE;                            // Set move down
	                #sx_MoveSectionUp := FALSE;                             // Reset move up
	            END_IF;

	            IF #sx_DivertUpRunTimeErr                                   // It took too long to move up
	                AND #sx_MoveSectionDown                                 // It took too long to move down
	            THEN
	                #sx_MoveSectionDown := FALSE;
	            END_IF;
	        END_IF;
	    END_REGION

	    REGION 2.2 - Set errors

	        // Runtime delay error
	        IF #sx_DivertUpRunTimeErr                                       // It took too long to move up
	            OR #sx_DivertDownRunTimeErr                                 // It took too long to move down
	        THEN

	            #qUDT_HMIStatus.Specific.ErrRuntime := TRUE;                // Set error runtime error
	        END_IF;

	        // Airpressure not ok
	        IF NOT #ix_AirPressureOk                                        // Airpressure is not signalling
	            AND (#sx_LeftRequest OR #sx_RightRequest)                   // If there is request to move to the left or right position
	        THEN
	            #qUDT_HMIStatus.Specific.ErrAirpressureNotOk := TRUE;       // Set error airpressure
	        END_IF;

	        // configuration errors
	        #ta_ConfigErr[1] := #iUDT_DivertConfiguration."Conveyor length" = 0;
	        #ta_ConfigErr[2] := #iUDT_DivertConfiguration.ParcelDefaultLength = 0;

	        #sx_ConfigurationError := #iUDT_DivertConfiguration.SizeDivert  // Set the configuration error bit (No status!!)
	        AND (#ta_ConfigErr[1] OR #ta_ConfigErr[2]);


	    END_REGION

	    REGION 2.3 - Warning

	        #qUDT_HMIStatus.Specific.WarnAirPressure := NOT #ix_AirPressureOk;  // Airpressure is not signalling

	    END_REGION


	    REGION 2.4 - Common Error

	        #sUDT_Status.Error := #qUDT_HMIStatus.Specific.ErrRuntime                              // Direction verification found the Direction fault, stop the parcel
	        OR #qUDT_HMIStatus.Specific.ErrAirpressureNotOk                     // Upper jam PEC detected WHILE going Up
	        OR #qUDT_HMIStatus.Specific.ErrOverrun                              // Parcel travelled too far to divert
	        OR #sx_ConfigurationError;                                          // Configuration error, check values

	    END_REGION

	    REGION 2.5 - Common Warning

	        #sUDT_Status.Warning := #qUDT_HMIStatus.Specific.WarnAirPressure;   // Airpressure is not signalling

	    END_REGION

	END_REGION

	REGION 3 - Check conditions to set Equipment ready

	    //Conditions to set bit sx_Ready to operate

	    #sx_Ready := NOT #sUDT_Status.Error                                 // Error present
	    AND #ix_SafetyOk                                                    // Safety signalling OK
	    AND #ix_24vOk                                                       // 24V signalling OK
	    AND #ix_400vOk;                                                     // 400v signalling OK

	END_REGION

	REGION 4 - Stop Equipment

	    // Conditions to stop conveyor
	    IF (#sF_TRIG_Jog.Q                                                  // Trigger when conveyor stops jogging by HMI
	        AND #sx_ManualModeActive)                                       // Manual mode is active

	        OR (NOT #iqUDT_EquipmentControl.Command.AutomaticOn             // Conveyor stops if the bit AutomaticOn from control block is false
	        AND NOT #sx_ManualModeActive)                                   // Manual mode active bit

	        OR (NOT #sx_Ready                                               // Bit conveyor ready to run in automatic mode
	        AND NOT #sx_ManualModeActive)                                   // Manual mode active

	        OR #sR_TRIG_ManualMode.Q                                        // Trigger when manual mode is set on
	        OR #sF_TRIG_ManualMode.Q                                        // Trigger when manual mode is set off

	        OR NOT #ix_SafetyOk

	    THEN
	        //  Order to stop VFD

	        #sx_AutomaticActive := FALSE;                                   // Automatic mode is disable

	    END_IF;

	END_REGION

	REGION 5 - Start

	    REGION 5.1 - Set Automatic active

	        // The conditions to set the bit "startReceived" are:
	        // - Divert not in manual mode.
	        // - Divert ready to run.
	        // - Bit AutomaticOn from control block must be on.
	        // - Bit start form control block on.

	        IF #iqUDT_EquipmentControl.Command.Start
	            AND #iqUDT_EquipmentControl.Command.AutomaticOn
	            AND NOT #sx_ManualModeActive
	            AND #sx_Ready
	        THEN
	            #sx_AutomaticActive := TRUE;                                // Diverter active automatic mode
	        END_IF;

	    END_REGION

	    REGION 5.2 - Restart request
	        #iqUDT_EquipmentControl.Request.RestartRequired := NOT #sx_AutomaticActive
	        AND NOT #sx_ManualModeActive
	        AND #sx_Ready;

	    END_REGION

	END_REGION

	REGION 6 - Manual mode

	    REGION 6.1 - Manual mode force disable

	        // Manual mode bits inputs can be reset in case of malfunction
	        IF #iqUDT_EquipmentControl.Command.DisableManualMode
	        THEN
	            #iqUDT_DivertCommand.ManualMode := FALSE;
	            #iqUDT_EquipmentControl.Command.ManualMode := False;
	        END_IF;

	    END_REGION

	    REGION 6.2 - Manual mode activation

	        // Manual mode is active if it is active from hmi or by control block
	        #sx_ManualModeActive := #iqUDT_EquipmentControl.Command.ManualMode
	        OR #iqUDT_DivertCommand.ManualMode;

	    END_REGION

	    REGION 6.3 - Reset manual commands
	        //When the system is not any more in manual mode or when fatal error occurs the HMI commands should be reset
	        IF NOT #ix_SafetyOk
	            OR NOT #ix_24vOk                                            // 24V error status
	            OR NOT #ix_400vOk                                           // 400V error status
	            OR NOT #ix_HardwareOk                                       // Profinet error status
	            OR NOT #sx_ManualModeActive
	        THEN
	            #iqUDT_DivertCommand.ManualDown := FALSE;
	            #iqUDT_DivertCommand.ManualUp := FALSE;

	        END_IF;

	    END_REGION

	    REGION 6.4 - Start/Stop

	        // Pre start conditions to run in manual mode
	        #sx_PreStartManual := #sx_ManualModeActive                      // Manual mode active bit
	        AND #ix_SafetyOk                                                // Safety healthy bit
	        AND #ix_HardwareOk;                                             // Profinet comunication



	        #sR_TRIG_PrestartManual(CLK := #sx_PreStartManual);
	        // If manual command is active to one side, first button ha sto be released to accept new
	        #sx_ManUP := (#sR_TRIG_ManualGoUp.Q AND NOT #sx_ManDown) OR
	        (#sx_ManUP AND #iqUDT_DivertCommand.ManualUp);

	        #sx_ManDown := (#sR_TRIG_ManualGoDown.Q AND NOT #sx_ManUP) OR
	        (#sx_ManDown AND #iqUDT_DivertCommand.ManualDown);

	        // Do signal request (horn sounding before movement)
	        IF #sx_PreStartManual                                           // Pre start conditions to run in manual mode
	            AND (#sR_TRIG_ManualGoUp.Q AND #sx_ManUP)                   // Trigger when conveyor start running in manual mode
	            OR (#sR_TRIG_ManualGoDown.Q AND #sx_ManDown)
	        THEN

	            #iqUDT_EquipmentControl.Request.SignalingRequest := TRUE;   // Request signaling to control block before conveyor run in manual mode

	        END_IF;

	        // Go up in manual mode
	        #sx_ManualGoUp := #sx_PreStartManual                            // Pre start conditions to run in manual mode
	        AND (NOT #iqUDT_EquipmentControl.Request.SignalingRequest       // Signaling request done
	        OR #sx_ManualRunning)
	        AND #sx_ManUP;                                                  // Manual mode start TO run

	        // Go down in manual mode
	        #sx_ManualGoDown := #sx_PreStartManual                          // Pre start conditions to run in manual mode
	        AND (NOT #iqUDT_EquipmentControl.Request.SignalingRequest       // Signaling request done
	        OR #sx_ManualRunning)
	        AND #sx_ManDown;                                                // Manual mode start to run

	        #sx_ManualRunning := #sx_ManualGoUp
	        OR #sx_ManualGoDown;

	    END_REGION
	END_REGION

	REGION 7 - Automatic mode

	    REGION 7.1 - Direction from decision point
	        IF #iqi_RequestedPosition <> 0 AND NOT (#sx_LeftRequest OR #sx_RightRequest)                                 // Position is received from decision block
	        THEN
	            #si_Direction := #iqi_RequestedPosition;                    // Copy the input to the memory
	            #si_Gin := #ii_Gin;                                         // Copy the found GIN number
	            #si_OldDirection := #si_Direction;
	            // As we found a divert decision we need to calculate the divert position if its based on position and not time
	            //
	            IF #iUDT_DivertConfiguration.SizeDivert
	            THEN
	                // Divert position is center of the divert section + half of the parcel.
	                //
	                #si_length := "DB_GIN".GIN[#si_Gin].General.Length;
	                IF #si_length <= 0 THEN
	                    #si_length := #iUDT_DivertConfiguration.ParcelDefaultLength;
	                END_IF;

	                // Use dimension of parcel in GIN record
	                #sdi_Divertposition := (((#iUDT_DivertConfiguration."Conveyor length" / 10) - (#si_length)) / 2) + #iUDT_DivertConfiguration.PositionOffset;

	            END_IF;

	            #iqi_RequestedPosition := 0;                                // Reset requested position again as all is handled

	        END_IF;
	    END_REGION

	    REGION 7.2 - Position left / right / straight on
	        // 1 = Left, 2 = Right and 99 = Default
	        //
	        IF #si_Direction = 1                                            // If the position "left" is equal to the request
	            AND #sx_Ready                                               // Ready to operate, No errors active
	            AND #sx_AutomaticActive                                     // Automaticly started
	        THEN
	            #sx_RightRequest := FALSE;                                  // Reset right command
	            #sx_LeftRequest := TRUE;                                    // Set left command
	            #si_Position := 0;                                          // Reset position
	            #si_Direction := 0;                                         // Reset the memory
	        END_IF;

	        IF #si_Direction = 2                                            // If the position "right" is equal to the request
	            AND #sx_Ready                                               // Ready to operate, No errors active
	            AND #sx_AutomaticActive                                     // Automaticly started
	        THEN
	            #sx_RightRequest := TRUE;                                   // Set right command
	            #sx_LeftRequest := FALSE;                                   // Reset left command
	            #si_Position := 0;                                          // Reset position
	            #si_Direction := 0;                                         // Reset the memory
	        END_IF;

	        IF #si_Direction = 99                                           // If the position "straight" is equal to the request
	            AND #sx_Ready                                               // Ready to operate, No errors active
	            AND #sx_AutomaticActive                                     // Automaticly started
	        THEN
	            #si_Direction := 0;                                         // Reset the memory
	        END_IF;
	    END_REGION

	    REGION 7.3 - Sequence
	        REGION 7.3.1 - Sequence step 1: move up

	            // Once decided to go left or right the diverter has to move to upper position when the parcel is in divert position

	            IF #sx_AutomaticActive                                      // The divert is automaticly started
	                AND #sx_Ready                                           // Ready to run / no errors
	                AND (#sx_LeftRequest OR #sx_RightRequest)               // If there is request to move to the left or right position
	                AND NOT #ix_SectionIsUp                                 // And not in upper position
	                AND NOT #sx_Active                                      // Sequence is not yet activated
	                AND ((NOT #iUDT_DivertConfiguration.SizeDivert          // Not diverting on parcel size but on PEC
	                AND (#si_Position >= #iUDT_DivertConfiguration.LengthIn)) // NOT diverting on parcel size but on PEC
	                OR (#iUDT_DivertConfiguration.SizeDivert                // Diverting on parcel size
	                AND (#iqa_TrackingMainData[#sdi_Divertposition] = #si_Gin
	                AND #iqa_TrackingMainData[#sdi_Divertposition] <> 0))  // GIN at divertposition
	                OR (#si_Position >= #iUDT_DivertConfiguration."Conveyor length"))
	            THEN
	                #sx_Active := TRUE;                                 // Sequence is activated
	                #sx_MoveSectionUp := TRUE;                          // Set position to be 1 = Up
	            END_IF;

	            IF #sx_AutomaticActive                                      // The divert is automaticly started
	                AND #sx_Ready                                           // Ready to run / no errors
	                AND (#sx_LeftRequest OR #sx_RightRequest)               // If there is request to move to the left or right position
	                AND NOT #ix_SectionIsUp                                 // And not in upper position
	                AND NOT #sx_Active                                      // Sequence is not yet activated
	                AND ((#si_Position >= #iUDT_DivertConfiguration."Conveyor length")
	                )
	            THEN
	                #qUDT_HMIStatus.Specific.ErrOverrun := True;        // Set error, parcel went too far and can not be deverted (Stop main conveyor)
	                #sx_MoveSectionDown := FALSE;                           // Reset move down
	                #sx_LeftRequest := FALSE;                               // Reset requests fom position
	                #sx_RightRequest := FALSE;                              // Reset requests fom position
	                #sx_Active := FALSE;                                    // End of sequence
	            END_IF;
	        END_REGION

	        REGION 7.3.2 - Sequence step 2: start transport in desired direction

	            // As the divert is up, the transport will start

	            IF #sx_AutomaticActive                                      // The divert is automaticly started
	                AND #sx_Ready                                           // Ready to run / no errors
	                AND #sx_MoveSectionUp                                   // Step move section up
	                AND #ix_SectionIsUp                                     // And in upper position
	            THEN

	                FILL_BLK(IN := 0,                                       // Clear tracking area for divert on main conveyor
	                         COUNT := DINT_TO_ULINT(#iUDT_DivertConfiguration."Conveyor length" / 10),
	                         OUT => #iqa_TrackingMainData[0]);

	                #sx_TransportActive := TRUE;                            // Set transport
	                #sx_MoveSectionUp := FALSE;                             // Reset move up
	                #si_Position := 0;                                      // Reset position

	            END_IF;
	        END_REGION

	        REGION 7.3.3 - Sequence step 3: Parcel transport finished, move down

	            // The transport has cleared the photoeye on the downstream conveyor, move down

	            IF #sx_AutomaticActive                                      // The divert is automaticly started
	                AND #sx_Ready                                           // Ready to run / no errors
	                AND #sx_TransportActive                                 // Step transport parcel
	                AND ((NOT #iUDT_DivertConfiguration.SizeDivert          // Not diverting on parcel size but on PEC
	                AND (#si_Position >= #iUDT_DivertConfiguration.LengthOut)) // NOT diverting on parcel size but on PEC
	                OR
	                (#iUDT_DivertConfiguration.SizeDivert                   // Diverting on parcel size
	                AND ((#sx_LeftRequest AND #sR_TRIG_PECLeft.Q)           // Active transport to left, parcel cleared PEC
	                OR (#sx_RightRequest AND #sR_TRIG_PECRight.Q))          // Active transport to right, parcel cleared PEC
	                OR (#si_Position >= #iUDT_DivertConfiguration.LengthOut)))
	            THEN
	                #si_Gin := 0;                                           // Reset the GIN to write
	                #sx_MoveSectionDown := TRUE;                            // Set move down
	                #sx_TransportActive := FALSE;                           // Reset transport

	            END_IF;
	        END_REGION

	        REGION 7.3.4 - Sequence step 4: Divert is down

	            // The divert is down now reset requests

	            IF #sx_AutomaticActive                                      // The divert is automaticly started
	                AND #sx_Ready                                           // Ready to run / no errors
	                AND #sx_MoveSectionDown                                 // Step transport parcel
	                AND #ix_SectionIsDown
	            THEN
	                #sx_MoveSectionDown := FALSE;                           // Reset move down
	                #sx_LeftRequest := FALSE;                               // Reset requests fom position
	                #sx_RightRequest := FALSE;                              // Reset requests fom position
	                #sx_Active := FALSE;                                    // End of sequence
	            END_IF;
	        END_REGION
	    END_REGION

	    REGION 7.4 - Calculate position
	        // When transport is active displacement is added to position counter

	        IF NOT #sx_PECTriggerFiltered
	            AND (#sx_LeftRequest OR #sx_RightRequest)
	            AND (#qUDT_LowerConveyorInterface.RunFwd OR #qUDT_LowerConveyorInterface.RunRvs)
	        THEN
	            #si_Position += ABS(#ii_DisplacementLower);
	        END_IF;

	        IF #sx_PECTriggerFiltered
	            AND (#qUDT_UpperConveyorInterface.RunFwd OR #qUDT_UpperConveyorInterface.RunRvs)
	        THEN
	            #si_Position += ABS(#ii_DisplacementUpper);
	        END_IF;
	    END_REGION
	END_REGION

	REGION 8 - Outputs
	    // Statement section REGION

	    REGION 8.1 - Lifting device

	        #qx_SectionDown := (#sx_AutomaticActive AND (#sx_MoveSectionDown OR (NOT #sx_Active AND NOT #ix_SectionIsDown))
	        OR (#sx_ManualModeActive AND #sx_ManualGoDown));
	        #qx_SectionUp := (#sx_AutomaticActive AND #sx_MoveSectionUp)
	        OR (#sx_ManualModeActive AND #sx_ManualGoUp);

	    END_REGION

	    REGION 8.2 - Rollerconveyor

	        // Conveyor receives always RTR signal to run
	        #iqUDT_HandShakeLowerConveyor.RTR := TRUE;

	        // Run forward
	        //
	        #qUDT_LowerConveyorInterface.RunFwd := #sx_AutomaticActive
	        AND NOT #sx_Active
	        AND #ix_SectionIsDown;

	        // Hold signal to conveyor
	        #qUDT_LowerConveyorInterface.Hold := NOT #qUDT_LowerConveyorInterface.RunFwd AND NOT #qUDT_LowerConveyorInterface.RunRvs;

	    END_REGION

	    REGION 8.3 - Divert belt conveyor
	        // Conveyor running to left
	        #qUDT_UpperConveyorInterface.RunFwd := #sx_AutomaticActive
	        AND #sx_LeftRequest
	        AND #iqUDT_HandShakeLeftConveyor.RTR
	        AND #sx_TransportActive;

	        // Conveyor running to right
	        #qUDT_UpperConveyorInterface.RunRvs := #sx_AutomaticActive
	        AND #sx_RightRequest
	        AND #iqUDT_HandShakerightConveyor.RTR
	        AND #sx_TransportActive;

	        // Hold signal to conveyor
	        #qUDT_UpperConveyorInterface.Hold := NOT #qUDT_UpperConveyorInterface.RunFwd AND NOT #qUDT_UpperConveyorInterface.RunRvs;
	    END_REGION

	    REGION 8.3 - handshake outfeed conveyors

	        // Outfeed conveyor left side
	        #iqUDT_HandShakeLeftConveyor.RTS := #sx_TransportActive AND #sx_LeftRequest;
	        #iqUDT_HandShakeLeftConveyor.TIP := #qUDT_UpperConveyorInterface.RunFwd;
	        IF #iqUDT_HandShakeLeftConveyor.RTS
	        THEN
	            #iqUDT_HandShakeLeftConveyor.GIN := #si_Gin;
	            #iqUDT_HandShakeLeftConveyor.NrOfPosToShift := 1;
	        ELSE
	            #iqUDT_HandShakeLeftConveyor.GIN := 0;
	            #iqUDT_HandShakeLeftConveyor.NrOfPosToShift := 0;
	        END_IF;

	        // Outfeed conveyor right side

	        #iqUDT_HandShakerightConveyor.RTS := #sx_TransportActive AND #sx_RightRequest;
	        #iqUDT_HandShakerightConveyor.TIP := #qUDT_UpperConveyorInterface.RunFwd;
	        IF #iqUDT_HandShakerightConveyor.RTS
	        THEN
	            #iqUDT_HandShakerightConveyor.GIN := #si_Gin;
	            #iqUDT_HandShakerightConveyor.NrOfPosToShift := 1;
	        ELSE
	            #iqUDT_HandShakerightConveyor.GIN := 0;
	            #iqUDT_HandShakerightConveyor.NrOfPosToShift := 0;
	        END_IF;
	    END_REGION
	END_REGION

	REGION 9 - Statistics

	    REGION 9.1 - Device up time

	        IF #sx_UpTime OR #iqUDT_EquipmentControl.Command.ResetData                          // Reset statistics
	        THEN

	            "FC_Statistics"(ix_Reset := #iqUDT_EquipmentControl.Command.ResetData, // Reset statistics input
	                            ix_Activate := #sx_UpTime,
	                            ix_RTrigActivate := #sR_TRIG_DeviceUpTime.Q,                   // Statistics active trigger
	                            iqUDT_Statistics := #iqUDT_Statistics.ConveyorUp);             // Statistics values output

	        END_IF;

	    END_REGION

	    REGION 9.2 - Device down time

	        // Conveyor down is when conveyor is not in manual mode and has an error
	        IF #sx_DownTime OR #iqUDT_EquipmentControl.Command.ResetData OR #sUDT_Status.SafetyStop     // Reset statistics
	        THEN

	            "FC_Statistics"(ix_Reset := #iqUDT_EquipmentControl.Command.ResetData, // Reset statistics input
	                            ix_Activate := #sx_DownTime OR #sUDT_Status.SafetyStop,   // Activate statistics functions input
	                            ix_RTrigActivate := #sR_TRIG_DeviceDownTime.Q,                 // Statistics active trigger
	                            iqUDT_Statistics := #iqUDT_Statistics.ConveyorDown);           // Statistics values output

	        END_IF;
	    END_REGION

	    REGION 9.3 - Device stop time

	        IF #sx_StoppedTime OR #iqUDT_EquipmentControl.Command.ResetData                     // Reset statistics
	        THEN

	            "FC_Statistics"(ix_Reset := #iqUDT_EquipmentControl.Command.ResetData, // Reset statistics input
	                            ix_Activate := #sx_StoppedTime,                           // Activate statistics functions input
	                            ix_RTrigActivate := #sR_TRIG_DeviceStopped.Q,                  // Statistics active trigger
	                            iqUDT_Statistics := #iqUDT_Statistics.ConveyorStop);           // Statistics values output

	        END_IF;
	    END_REGION
	END_REGION





END_FUNCTION_BLOCK

FUNCTION_BLOCK "FB_CrossOver"
TITLE = FB_CrossOver
{ S7_Optimized_Access := 'TRUE' }
VERSION : 0.1
// ATTRIBUTES
// AUTO_NUMBER = True
// BLOCK_NUMBER = 196
// END_ATTRIBUTES
//Function to control a merge left/right/straight. A conveyor, part of the merge, will move up or down to change the direction. Moving up and down control is done by this block.
   VAR_INPUT
      iUDT_Configuration { ExternalAccessible := 'False'; ExternalVisible := 'False'; ExternalWritable := 'False'} : "UDT_CrossoverConfiguration";   // Configuration structure
      ii_DisplacementRoller { ExternalAccessible := 'False'; ExternalVisible := 'False'; ExternalWritable := 'False'} : Int;   // Actual displacement of the rollerconveyor
      ii_DisplacementBelt { ExternalAccessible := 'False'; ExternalVisible := 'False'; ExternalWritable := 'False'} : Int;   // Actual displacement of the beltconveyor
      ix_HardwareOk { ExternalAccessible := 'False'; ExternalVisible := 'False'; ExternalWritable := 'False'} : Bool;   // TRUE when  hardware is Ok
      ix_400vOk { ExternalAccessible := 'False'; ExternalVisible := 'False'; ExternalWritable := 'False'} : Bool;   // TRUE when 400VAC is healthy
      ix_24vOk { ExternalAccessible := 'False'; ExternalVisible := 'False'; ExternalWritable := 'False'} : Bool;   // TRUE when 24VDC is healthy
      ix_SafetyOk { ExternalAccessible := 'False'; ExternalVisible := 'False'; ExternalWritable := 'False'} : Bool;   // TRUE when safety is ok
      ix_AirPressureOk { ExternalAccessible := 'False'; ExternalVisible := 'False'; ExternalWritable := 'False'} : Bool;   // Air pressure circuit healthy
      ix_SectionIsDown { ExternalAccessible := 'False'; ExternalVisible := 'False'; ExternalWritable := 'False'} : Bool;   // TRUE when section is down
      ix_SectionIsUp { ExternalAccessible := 'False'; ExternalVisible := 'False'; ExternalWritable := 'False'} : Bool;   // TRUE when section is up
      ix_Conveyor1Auto { ExternalAccessible := 'False'; ExternalVisible := 'False'; ExternalWritable := 'False'} : Bool;   // Conveyor is started in auto
      ix_Conveyor2Auto { ExternalAccessible := 'False'; ExternalVisible := 'False'; ExternalWritable := 'False'} : Bool;   // Conveyor is started in auto
      ix_Conveyor3Auto { ExternalAccessible := 'False'; ExternalVisible := 'False'; ExternalWritable := 'False'} : Bool;   // Conveyor is started in auto
      ix_Conveyor4Auto { ExternalAccessible := 'False'; ExternalVisible := 'False'; ExternalWritable := 'False'} : Bool;   // Conveyor is started in auto
      ix_PECOutfeed { ExternalAccessible := 'False'; ExternalVisible := 'False'; ExternalWritable := 'False'} : Bool;   // True when outfeed PEC is not occupied
   END_VAR

   VAR_OUTPUT
      qUDT_HMIStatus { ExternalAccessible := 'False'; ExternalVisible := 'False'; ExternalWritable := 'False'} : "UDT_Crossoverstatus";   // HMI status structure
      qUDT_Status { ExternalAccessible := 'False'; ExternalVisible := 'False'; ExternalWritable := 'False'} : "UDT_CommonStatus";   // Common status structure
      qUDT_RollerConveyorInterface { ExternalAccessible := 'False'; ExternalVisible := 'False'; ExternalWritable := 'False'} : Struct   // Interface roller conveyor
         Hold { ExternalAccessible := 'False'; ExternalVisible := 'False'; ExternalWritable := 'False'} : Bool;   // Hold the conveyor
         RunFwd { ExternalAccessible := 'False'; ExternalVisible := 'False'; ExternalWritable := 'False'} : Bool;   // Run conveyor forward
         RunRvs { ExternalAccessible := 'False'; ExternalVisible := 'False'; ExternalWritable := 'False'} : Bool;   // Run conveyor reverse
      END_STRUCT;
      qUDT_BeltConveyorInterface { ExternalAccessible := 'False'; ExternalVisible := 'False'; ExternalWritable := 'False'} : Struct   // Interface belt conveyor
         Hold { ExternalAccessible := 'False'; ExternalVisible := 'False'; ExternalWritable := 'False'} : Bool;   // Hold the conveyor
         RunFwd { ExternalAccessible := 'False'; ExternalVisible := 'False'; ExternalWritable := 'False'} : Bool;   // Run conveyor forward
         RunRvs { ExternalAccessible := 'False'; ExternalVisible := 'False'; ExternalWritable := 'False'} : Bool;   // Run conveyor reverse
      END_STRUCT;
      qx_SectionUp { ExternalAccessible := 'False'; ExternalVisible := 'False'; ExternalWritable := 'False'} : Bool;   // Output to control section up
      qx_SectionDown { ExternalAccessible := 'False'; ExternalVisible := 'False'; ExternalWritable := 'False'} : Bool;   // Output to control section down
   END_VAR

   VAR_IN_OUT
      iqa_TrackingDataRoller : Array[*] of Int;   // Tracking data
      iqa_TrackingDataBelt : Array[*] of Int;   // Tracking data
      iqUDT_EquipmentControl : "UDT_EquipmentControl";   // Equipment control structure
      iqUDT_CrossOverCommand : "UDT_CrossoverCommand";   // Conveyor command stucture
      iqUDT_Statistics : "UDT_ConveyorStatistics";   // Statistics structure
      iqUDT_HandShakeRollerConveyor : "UDT_ConveyorHandshake";
      iqUDT_HandShakeBeltConveyor : "UDT_ConveyorHandshake";
      iqUDT_HandShakeConveyor1 : "UDT_ConveyorHandshake";   // Handshake structure low level conveyor
      iqUDT_HandShakeConveyor2 : "UDT_ConveyorHandshake";   // Handshake structure low level conveyor
      iqUDT_HandShakeConveyor3 : "UDT_ConveyorHandshake";   // Handshake structure high level conveyor
      iqUDT_HandShakeConveyor4 : "UDT_ConveyorHandshake";   // Handshake structure high level conveyor
   END_VAR

   VAR
      sa_FiFo { ExternalAccessible := 'False'; ExternalVisible := 'False'; ExternalWritable := 'False'} : Array[1..#ci_FiFoLength] of Int;   // FiFo for
      sUDT_Status { ExternalAccessible := 'False'; ExternalVisible := 'False'; ExternalWritable := 'False'; S7_SetPoint := 'False'} : "UDT_CommonStatus";   // Common status structure
      sUDT_StatusOld { ExternalAccessible := 'False'; ExternalVisible := 'False'; ExternalWritable := 'False'; S7_SetPoint := 'False'} : "UDT_CommonStatus";   // Common status structure
      sFB_UpMonitor { ExternalAccessible := 'False'; ExternalVisible := 'False'; ExternalWritable := 'False'; S7_SetPoint := 'False'} : "FB_TimerOnOffDelay";   // Timer to monitor divert took too long to move to upper position
      sFB_DownMonitor { ExternalAccessible := 'False'; ExternalVisible := 'False'; ExternalWritable := 'False'; S7_SetPoint := 'False'} : "FB_TimerOnOffDelay";
      sFB_PECOutfeedOnOffDelay { ExternalAccessible := 'False'; ExternalVisible := 'False'; ExternalWritable := 'False'; S7_SetPoint := 'False'} : "FB_TimerOnOffDelay";
      sR_TRIG_RTSConveyor1 {InstructionName := 'R_TRIG'; LibVersion := '1.0'; ExternalAccessible := 'False'; ExternalVisible := 'False'; ExternalWritable := 'False'; S7_SetPoint := 'False'} : R_TRIG;   // Rising edge trigger RTS signal from infeed
      sR_TRIG_RTSConveyor2 {InstructionName := 'R_TRIG'; LibVersion := '1.0'; ExternalAccessible := 'False'; ExternalVisible := 'False'; ExternalWritable := 'False'; S7_SetPoint := 'False'} : R_TRIG;   // Rising edge trigger RTS signal from infeed
      sR_TRIG_RTSConveyor3 {InstructionName := 'R_TRIG'; LibVersion := '1.0'; ExternalAccessible := 'False'; ExternalVisible := 'False'; ExternalWritable := 'False'; S7_SetPoint := 'False'} : R_TRIG;   // Rising edge trigger RTS signal from infeed
      sR_TRIG_RTSConveyor4 {InstructionName := 'R_TRIG'; LibVersion := '1.0'; ExternalAccessible := 'False'; ExternalVisible := 'False'; ExternalWritable := 'False'; S7_SetPoint := 'False'} : R_TRIG;   // Rising edge trigger RTS signal from infeed
      sF_TRIG_Transport {InstructionName := 'F_TRIG'; LibVersion := '1.0'; ExternalAccessible := 'False'; ExternalVisible := 'False'; ExternalWritable := 'False'; S7_SetPoint := 'False'} : F_TRIG;   // Falling edge trigger transport
      sR_TRIG_ManualMode {InstructionName := 'R_TRIG'; LibVersion := '1.0'; ExternalAccessible := 'False'; ExternalVisible := 'False'; ExternalWritable := 'False'; S7_SetPoint := 'False'} : R_TRIG;   // Rising edge trigger manual mode
      sF_TRIG_ManualMode {InstructionName := 'F_TRIG'; LibVersion := '1.0'; ExternalAccessible := 'False'; ExternalVisible := 'False'; ExternalWritable := 'False'; S7_SetPoint := 'False'} : F_TRIG;   // Falling edge trigger manual mode
      sR_TRIG_PrestartManual {InstructionName := 'R_TRIG'; LibVersion := '1.0'; ExternalAccessible := 'False'; ExternalVisible := 'False'; ExternalWritable := 'False'; S7_SetPoint := 'False'} : R_TRIG;   // Rising edge of manual prestart
      sR_TRIG_ManualGoUp {InstructionName := 'R_TRIG'; LibVersion := '1.0'; ExternalAccessible := 'False'; ExternalVisible := 'False'; ExternalWritable := 'False'; S7_SetPoint := 'False'} : R_TRIG;   // Rising edge run conveyor in manual mode
      sR_TRIG_ManualGoDown {InstructionName := 'R_TRIG'; LibVersion := '1.0'; ExternalAccessible := 'False'; ExternalVisible := 'False'; ExternalWritable := 'False'; S7_SetPoint := 'False'} : R_TRIG;   // Rising edge trigger manual jog
      sR_TRIG_PecOutfeed {InstructionName := 'R_TRIG'; LibVersion := '1.0'; ExternalAccessible := 'False'; ExternalVisible := 'False'; ExternalWritable := 'False'; S7_SetPoint := 'False'} : R_TRIG;   // Rising edge of reverse direction
      sF_TRIG_Jog {InstructionName := 'F_TRIG'; LibVersion := '1.0'; ExternalAccessible := 'False'; ExternalVisible := 'False'; ExternalWritable := 'False'; S7_SetPoint := 'False'} : F_TRIG;   // Falling edge trigger manual mode jog
      sR_TRIG_DeviceUpTime {InstructionName := 'R_TRIG'; LibVersion := '1.0'; ExternalAccessible := 'False'; ExternalVisible := 'False'; ExternalWritable := 'False'; S7_SetPoint := 'False'} : R_TRIG;   // Rising edge trigger conveyor up time
      sR_TRIG_DeviceStopped {InstructionName := 'R_TRIG'; LibVersion := '1.0'; ExternalAccessible := 'False'; ExternalVisible := 'False'; ExternalWritable := 'False'; S7_SetPoint := 'False'} : R_TRIG;   // Rising edge of stop
      sR_TRIG_DeviceDownTime {InstructionName := 'R_TRIG'; LibVersion := '1.0'; ExternalAccessible := 'False'; ExternalVisible := 'False'; ExternalWritable := 'False'; S7_SetPoint := 'False'} : R_TRIG;   // Rising edge trigger conveyor down
      si_Step { ExternalAccessible := 'False'; ExternalVisible := 'False'; ExternalWritable := 'False'} : Int;
      si_Conveyor { ExternalAccessible := 'False'; ExternalVisible := 'False'; ExternalWritable := 'False'} : Int;   // Active infeed
      si_LoopArrayCount { ExternalAccessible := 'False'; ExternalVisible := 'False'; ExternalWritable := 'False'} : Int;   // FiFo process counter
      si_Gin { ExternalAccessible := 'False'; ExternalVisible := 'False'; ExternalWritable := 'False'} : Int;   // New GIN found
      si_Length { ExternalAccessible := 'False'; ExternalVisible := 'False'; ExternalWritable := 'False'} : Int;   // Length of the product
      si_Stopposition { ExternalAccessible := 'False'; ExternalVisible := 'False'; ExternalWritable := 'False'} : Int;   // Position to stop
      si_Position { ExternalAccessible := 'False'; ExternalVisible := 'False'; ExternalWritable := 'False'} : Int;   // Position counter
      sx_PECOutfeedFiltered { ExternalAccessible := 'False'; ExternalVisible := 'False'; ExternalWritable := 'False'} : Bool;   // Signal filtered with on and off delay
      sx_PECLeftFiltered { ExternalAccessible := 'False'; ExternalVisible := 'False'; ExternalWritable := 'False'} : Bool;   // Signal filtered with on and off delay
      sx_PECRightFiltered { ExternalAccessible := 'False'; ExternalVisible := 'False'; ExternalWritable := 'False'} : Bool;   // Signal filtered with on and off delay
      sx_Active { ExternalAccessible := 'False'; ExternalVisible := 'False'; ExternalWritable := 'False'} : Bool;   // Device sequence is activated for parcel
      sx_DataReceived { ExternalAccessible := 'False'; ExternalVisible := 'False'; ExternalWritable := 'False'} : Bool;   // Handshake from upstream conveyor
      sx_InfeedCHK { ExternalAccessible := 'False'; ExternalVisible := 'False'; ExternalWritable := 'False'} : Bool;   // Step Infeed check
      sx_MoveSectionUpinfeed { ExternalAccessible := 'False'; ExternalVisible := 'False'; ExternalWritable := 'False'} : Bool;   // Step move device to upper position
      sx_MoveSectionUpOutfeed { ExternalAccessible := 'False'; ExternalVisible := 'False'; ExternalWritable := 'False'} : Bool;   // Step move device to upper position
      sx_MoveSectionUpEnd { ExternalAccessible := 'False'; ExternalVisible := 'False'; ExternalWritable := 'False'} : Bool;   // Step move device to upper position
      sx_MoveSectionDownInfeed { ExternalAccessible := 'False'; ExternalVisible := 'False'; ExternalWritable := 'False'} : Bool;   // Step move device to lower position
      sx_MoveSectionDownOutfeed { ExternalAccessible := 'False'; ExternalVisible := 'False'; ExternalWritable := 'False'} : Bool;   // Step move device to lower position
      sx_MoveSectiondownEnd { ExternalAccessible := 'False'; ExternalVisible := 'False'; ExternalWritable := 'False'} : Bool;   // Step move device to lower position
      sx_BeltTransportIn { ExternalAccessible := 'False'; ExternalVisible := 'False'; ExternalWritable := 'False'} : Bool;   // Step transport is activated
      sx_BeltTransportOut { ExternalAccessible := 'False'; ExternalVisible := 'False'; ExternalWritable := 'False'} : Bool;   // Step transport is activated
      sx_RollerTransportIn { ExternalAccessible := 'False'; ExternalVisible := 'False'; ExternalWritable := 'False'} : Bool;   // Step transport is activated
      sx_RollerTransportOut { ExternalAccessible := 'False'; ExternalVisible := 'False'; ExternalWritable := 'False'} : Bool;   // Step transport is activated
      sx_RollerRTR { ExternalAccessible := 'False'; ExternalVisible := 'False'; ExternalWritable := 'False'} : Bool;   // Lower deck RTR signal
      sx_BeltRTR { ExternalAccessible := 'False'; ExternalVisible := 'False'; ExternalWritable := 'False'} : Bool;   // Upper deck RTR signal
      sx_Ready { ExternalAccessible := 'False'; ExternalVisible := 'False'; ExternalWritable := 'False'} : Bool;   // Conveyor Ready to operate in Automatic mode
      sx_AutomaticActive { ExternalAccessible := 'False'; ExternalVisible := 'False'; ExternalWritable := 'False'} : Bool;   // Running in automatic
      sx_PreStartManual { ExternalAccessible := 'False'; ExternalVisible := 'False'; ExternalWritable := 'False'} : Bool;   // Pre conditions to run conveyor in manual mode
      sx_ManualModeActive { ExternalAccessible := 'False'; ExternalVisible := 'False'; ExternalWritable := 'False'} : Bool;   // Manual mode active
      sx_ManualRunning { ExternalAccessible := 'False'; ExternalVisible := 'False'; ExternalWritable := 'False'} : Bool;   // Conveyor running in manual mode
      sx_ManualGoUp { ExternalAccessible := 'False'; ExternalVisible := 'False'; ExternalWritable := 'False'} : Bool;   // Manual control go Up
      sx_ManualGoDown { ExternalAccessible := 'False'; ExternalVisible := 'False'; ExternalWritable := 'False'} : Bool;   // Manual control go down
      sx_ManUP { ExternalAccessible := 'False'; ExternalVisible := 'False'; ExternalWritable := 'False'} : Bool;   // Manual go up
      sx_ManDown { ExternalAccessible := 'False'; ExternalVisible := 'False'; ExternalWritable := 'False'} : Bool;   // Manual go down
      sx_ConfigurationError { ExternalAccessible := 'False'; ExternalVisible := 'False'; ExternalWritable := 'False'} : Bool;   // Commissioning: configuration of parameters is wrong
      sx_OutfeedLowlevel { ExternalAccessible := 'False'; ExternalVisible := 'False'; ExternalWritable := 'False'} : Bool;   // The outfeedis low level
      sx_OutfeedHighlevel { ExternalAccessible := 'False'; ExternalVisible := 'False'; ExternalWritable := 'False'} : Bool;   // The outfeedis high level
      sx_NoHighLevelInfeed { ExternalAccessible := 'False'; ExternalVisible := 'False'; ExternalWritable := 'False'} : Bool;   // None of the high level conveyors isinfeed
      sx_NoLowLevelInfeed { ExternalAccessible := 'False'; ExternalVisible := 'False'; ExternalWritable := 'False'} : Bool;   // None of the low level conveyors isinfeed
      sx_LeftRequest { ExternalAccessible := 'False'; ExternalVisible := 'False'; ExternalWritable := 'False'} : Bool;   // Request left outfeed position for actual parcel
      sx_RightRequest { ExternalAccessible := 'False'; ExternalVisible := 'False'; ExternalWritable := 'False'} : Bool;   // Request right outfeed position for actual parcel
      sx_DivertUpRunTimeErr { ExternalAccessible := 'False'; ExternalVisible := 'False'; ExternalWritable := 'False'} : Bool;   // It is taking too long to move divert up
      sx_DivertDownRunTimeErr { ExternalAccessible := 'False'; ExternalVisible := 'False'; ExternalWritable := 'False'} : Bool;   // It is taking too long to move divert down
      sx_UpTime { ExternalAccessible := 'False'; ExternalVisible := 'False'; ExternalWritable := 'False'} : Bool;   // Device is up
      sx_DownTime { ExternalAccessible := 'False'; ExternalVisible := 'False'; ExternalWritable := 'False'} : Bool;   // Device is down
      sx_StoppedTime { ExternalAccessible := 'False'; ExternalVisible := 'False'; ExternalWritable := 'False'} : Bool;   // Device is stopped
   END_VAR

   VAR_TEMP
      ta_ConfigErr : Array[0..10] of Bool;
   END_VAR

   VAR CONSTANT
      ci_FiFoLength : Int := 10;
   END_VAR


BEGIN
	(*
	----------------------------------------------------------------------------------------

	Version history:
	Date        | Version   | Author        | Remark
	----------------------------------------------------------------------------------------
	01/03/2023  | 1.0       | F.Baten       | Initial version
	*)

	REGION 1 - Initial
	    REGION 1.1 - First PLC cycle

	        IF "DB_Memory".FirstScan
	        THEN
	            #sx_AutomaticActive := FALSE;                                       // switch of automatic activ

	        END_IF;

	    END_REGION

	    REGION 1.2 - Triggers

	        // Rising edge trigger manual mode
	        #sR_TRIG_ManualMode(CLK := #iqUDT_CrossOverCommand.ManualMode
	                            OR #iqUDT_EquipmentControl.Command.ManualMode);

	        // Falling edge trigger manual mode
	        #sF_TRIG_ManualMode(CLK := #iqUDT_CrossOverCommand.ManualMode
	                            OR #iqUDT_EquipmentControl.Command.ManualMode);

	        // Rising edge trigger to start in manual mode
	        #sR_TRIG_ManualGoUp(CLK := #iqUDT_CrossOverCommand.ManualUp);

	        // Rising edge trigger manual mode jog
	        #sR_TRIG_ManualGoDown(CLK := #iqUDT_CrossOverCommand.ManualDown);

	        // Rising edge PEC outfeed
	        #sR_TRIG_PecOutfeed(CLK := #sx_PECOutfeedFiltered);

	        // Infeed conveyor is ready to send
	        #sR_TRIG_RTSConveyor1(CLK := #iUDT_Configuration.Conveyor1.IsInfeed AND #iqUDT_HandShakeConveyor1.RTS AND #ix_Conveyor1Auto);
	        #sR_TRIG_RTSConveyor2(CLK := #iUDT_Configuration.Conveyor2.IsInfeed AND #iqUDT_HandShakeConveyor2.RTS AND #ix_Conveyor2Auto);
	        #sR_TRIG_RTSConveyor3(CLK := #iUDT_Configuration.Conveyor3.IsInfeed AND #iqUDT_HandShakeConveyor3.RTS AND #ix_Conveyor3Auto);
	        #sR_TRIG_RTSConveyor4(CLK := #iUDT_Configuration.Conveyor4.IsInfeed AND #iqUDT_HandShakeConveyor4.RTS AND #ix_Conveyor4Auto);

	        // Rising edge equipment uptime
	        #sR_TRIG_DeviceUpTime(CLK := #sx_UpTime);

	        //Rising edge equipment stopped
	        #sR_TRIG_DeviceStopped(CLK := #sx_StoppedTime);

	        // Rising edge equipment conveyor downtime
	        #sR_TRIG_DeviceDownTime(CLK := #sx_DownTime);
	    END_REGION

	    REGION 1.3 - Timers
	        // Statement section REGION
	        #sFB_PECOutfeedOnOffDelay(iudi_OnDelayTime := #iUDT_Configuration.OutfeedTimeOnDelay,         // Off delay time to filter PEC signal
	                                  iudi_OffDelayTime := #iUDT_Configuration.OutfeedTimeOffDelay,     // On delay time to filter PEC signal
	                                  ix_SignalToDelay := #ix_PECOutfeed,                               // PEC input signal
	                                  ix_Enable := TRUE,
	                                  qx_DelayedSignal => #sx_PECOutfeedFiltered);                      // PEC signal filtered

	        #sFB_UpMonitor(iudi_OnDelayTime := #iUDT_Configuration.LiftRuntimeUpOnDelay,                // Off delay time
	                       iudi_OffDelayTime := #iUDT_Configuration.LiftRuntimeUpOffDelay,              // On delay time
	                       ix_SignalToDelay := #sx_AutomaticActive
	                       AND #sx_MoveSectionUpinfeed
	                       AND NOT #ix_SectionIsUp,                                                     // input signal
	                       ix_Enable := TRUE,
	                       qx_DelayedSignal => #sx_DivertUpRunTimeErr);                                 // Signal filtered

